						(* 1720: Bandklemmen links *)
						zyl_bandklemmen_li.fb.st_config.b_config_fertig := FALSE;
						zyl_bandklemmen_li.fb.st_config.b_endlage1_aktiv := FALSE;
						zyl_bandklemmen_li.fb.st_config.b_endlage2_aktiv := FALSE;
						zyl_bandklemmen_li.fb.st_config.b_sensor1_aktiv := FALSE;
						zyl_bandklemmen_li.fb.st_config.b_sensor2_aktiv := FALSE;
						zyl_bandklemmen_li.fb.st_config.i16_gruppe := 1;
						zyl_bandklemmen_li.fb.st_config.i16_identnummer := 3;
						zyl_bandklemmen_li.fb.st_config.i16_meld_startindex := 2040;
						zyl_bandklemmen_li.fb.st_config.str_beschreibung := ' ';
						zyl_bandklemmen_li.fb.st_config.str_instanz_name := 'Bandklemmen links';
						zyl_bandklemmen_li.fb.st_config.str_zylinder_typ := '1V0E_NO';
						zyl_bandklemmen_li.fb.st_config.t_ein_aus_fahrzeit := t#0ms;
						zyl_bandklemmen_li.fb.st_config.t_ueberwachungszeit := t#500ms;
						zyl_bandklemmen_li.fb.st_config.i16_tzk_faktor_ausfahren := 100;
						zyl_bandklemmen_li.fb.st_config.i16_tzk_faktor_einfahren := 100;
						zyl_bandklemmen_li.fb.st_config.b_config_fertig := TRUE;
						(* 1720: Bandklemmen rechts *)
						zyl_bandklemmen_re.fb.st_config.b_config_fertig := FALSE;
						zyl_bandklemmen_re.fb.st_config.b_endlage1_aktiv := FALSE;
						zyl_bandklemmen_re.fb.st_config.b_endlage2_aktiv := FALSE;
						zyl_bandklemmen_re.fb.st_config.b_sensor1_aktiv := FALSE;
						zyl_bandklemmen_re.fb.st_config.b_sensor2_aktiv := FALSE;
						zyl_bandklemmen_re.fb.st_config.i16_gruppe := 1;
						zyl_bandklemmen_re.fb.st_config.i16_identnummer := 4;
						zyl_bandklemmen_re.fb.st_config.i16_meld_startindex := 2060;
						zyl_bandklemmen_re.fb.st_config.str_beschreibung := ' ';
						zyl_bandklemmen_re.fb.st_config.str_instanz_name := 'Bandklemmen rechts';
						zyl_bandklemmen_re.fb.st_config.str_zylinder_typ := '1V0E_NO';
						zyl_bandklemmen_re.fb.st_config.t_ein_aus_fahrzeit := t#0ms;
						zyl_bandklemmen_re.fb.st_config.t_ueberwachungszeit := t#500ms;
						zyl_bandklemmen_re.fb.st_config.i16_tzk_faktor_ausfahren := 100;
						zyl_bandklemmen_re.fb.st_config.i16_tzk_faktor_einfahren := 100;
						zyl_bandklemmen_re.fb.st_config.b_config_fertig := TRUE;
				
					BANDWECHSLER_V2:
						;

					SERVO:
						;
				END_CASE;
		ELSE
			b_config_fertig := FALSE;
		END_IF

	RASTERFOLIE:
		;
END_CASE
END_PROGRAM

(* POU Maschine1720/ST_Bandeinzug_Kontroller_1720, ST *)
PROGRAM ST_Bandeinzug_Kontroller_1720
VAR_INPUT
	st_config							: struct_config;
	st_ctrl_in							: struct_ctrl_in;
END_VAR
VAR_IN_OUT
	st_visu							: struct_visu;
END_VAR
VAR_OUTPUT
	st_ctrl_out						: struct_ctrl_out;
END_VAR
VAR
	fb_ton_wz						: TON;
	fb_ton_uez						: TON;
	fb_ton_quitt						: TON;
	fb_state_entry						: ST_StateEntry;
	e_ls_bandende_re				AT %I* : BOOL;
	e_ls_bandende_li					AT %I* : BOOL;

	fb_r_trig_vorschubkontrolle_li		: R_TRIG;
	fb_f_trig_vorschubkontrolle_li		: F_TRIG;
	fb_r_trig_nocke_einzug				: R_TRIG;
	fb_f_trig_nocke_einzug				: F_TRIG;
	b_hm_pos_flanke_vorschub_li		: BOOL := FALSE;
	b_hm_neg_flanke_vorschub_li		: BOOL := FALSE;
	sm_fehler_bandvorschub_li			: BOOL := FALSE;
	fb_r_trig_vorschubkontrolle_re		: R_TRIG;
	fb_f_trig_vorschubkontrolle_re		: F_TRIG;
	b_hm_pos_flanke_vorschub_re		: BOOL := FALSE;
	b_hm_neg_flanke_vorschub_re		: BOOL := FALSE;
	sm_fehler_bandvorschub_re			: BOOL := FALSE;
	sm_keine_busverbindung			: BOOL := FALSE;

	e_wc_state							AT %I* : BOOL;	(* 0=Data valid, 1=Data invalid *)
	e_gls_bandvorschubkontrolle_li		AT %I* : BOOL;
	e_gls_bandvorschubkontrolle_re		AT %I* : BOOL;
END_VAR
(* Zeiten *)
fb_ton_wz(IN:= , PT:= , Q=>  , ET=> );
fb_ton_uez(IN:= , PT:= , Q=>  , ET=> );
fb_ton_quitt(IN:= , PT:= t#100ms, Q=> , ET=> );

(* Flanken *)
fb_f_trig_vorschubkontrolle_li(CLK:= e_gls_bandvorschubkontrolle_li, Q=> );
fb_r_trig_vorschubkontrolle_li(CLK:= e_gls_bandvorschubkontrolle_li, Q=> );
fb_f_trig_nocke_einzug(CLK:= nockenschaltwerk_bestueckachse.fb.arr_spur[SP_PNEUMATIKBANDEINZUG_GLS], Q=> );
fb_r_trig_nocke_einzug(CLK:= nockenschaltwerk_bestueckachse.fb.arr_spur[SP_PNEUMATIKBANDEINZUG_GLS], Q=> );
fb_f_trig_vorschubkontrolle_re(CLK:= e_gls_bandvorschubkontrolle_re, Q=> );
fb_r_trig_vorschubkontrolle_re(CLK:= e_gls_bandvorschubkontrolle_re, Q=> );

(*neue Haltezylinder für Bandklemmeinzug*)
(*bei Steuerung Ein oben bei Steuerung Aus wird selbständig über Federkraft geklemmt*)
IF ST_Safetyprogramm.se_steuerung_ein THEN
	zyl_bawe_halter_li.st_ctrl.in.b_einfahren := TRUE;
	zyl_bawe_halter_re.st_ctrl.in.b_einfahren := TRUE;
END_IF

(* Toplevel *)
IF fb_state_entry.i16_next_step > INIT AND fb_state_entry.i16_next_step < FEHLER THEN
	IF fb_state_entry.i16_next_step < STOP THEN
		IF st_ctrl_in.b_stop THEN
			fb_state_entry.i16_next_step := STOP;
		END_IF
	END_IF
	(* Allgemeine Fehler *)
	IF	NOT gst_datensatz.st_md.b_wt_transport_simulation AND
		(zyl_bandfaenger_li.st_ctrl.out.b_fehler OR
		zyl_bandklemmen_li.st_ctrl.out.b_fehler OR
		zyl_bandfaenger_re.st_ctrl.out.b_fehler OR
		zyl_bandklemmen_re.st_ctrl.out.b_fehler OR
		zyl_bawe_halter_li.st_ctrl.out.b_fehler OR
		zyl_bawe_halter_re.st_ctrl.out.b_fehler)
		THEN
			fb_state_entry.i16_next_step := FEHLER;
	(* Zylinder im Handbetrieb *)
	ELSIF	 gi16_betriebsart = HAND AND (
			(st_visu.st_zyl.i16_nr_zyl_im_handbetrieb = zyl_bandfaenger_li.fb.st_config.i16_identnummer OR
			st_visu.st_zyl.i16_nr_zyl_im_handbetrieb = zyl_bandfaenger_li.fb.st_config.i16_identnummer OR
			st_visu.st_zyl.i16_nr_zyl_im_handbetrieb = zyl_bandfaenger_re.fb.st_config.i16_identnummer OR
			st_visu.st_zyl.i16_nr_zyl_im_handbetrieb = zyl_bandklemmen_re.fb.st_config.i16_identnummer OR
			st_visu.st_zyl.i16_nr_zyl_im_handbetrieb = zyl_bawe_halter_li.fb.st_config.i16_identnummer OR
			st_visu.st_zyl.i16_nr_zyl_im_handbetrieb = zyl_bawe_halter_re.fb.st_config.i16_identnummer))
			THEN
				fb_state_entry.i16_next_step := FEHLER;
	END_IF
END_IF

(* ======================================Schrittkette======================================== *)
fb_state_entry(
	i16_next_step:= ,
	i16_pos:= 1,
	s_debugtext:= ,
	E=> ,
	X=> , 
	i16_step=> ,
	i16_last_step=> );

CASE fb_state_entry.i16_step OF
(*=======================================================*)
	INIT_OBJ:
		IF st_config.b_config_fertig THEN
			fb_state_entry.i16_next_step := INIT;
		END_IF

(*=======================================================*)
	INIT:
		IF fb_state_entry.E THEN
			fb_ton_wz.IN := FALSE;
			fb_ton_uez.IN := FALSE;
			fb_ton_quitt.IN := FALSE;
			st_ctrl_out.b_fehler := FALSE;
			st_ctrl_out.b_bereit := FALSE;
			st_ctrl_out.b_fertig := FALSE;
			zyl_bandfaenger_li.st_ctrl.in.b_ausfahren := FALSE;
			zyl_bandfaenger_li.st_ctrl.in.b_einfahren := FALSE;
			 zyl_bandklemmen_li.st_ctrl.in.b_ausfahren := FALSE;
			 zyl_bandklemmen_li.st_ctrl.in.b_einfahren := FALSE;
			zyl_bandfaenger_re.st_ctrl.in.b_ausfahren := FALSE;
			zyl_bandfaenger_re.st_ctrl.in.b_einfahren := FALSE;
			 zyl_bandklemmen_re.st_ctrl.in.b_ausfahren := FALSE;
			 zyl_bandklemmen_re.st_ctrl.in.b_einfahren := FALSE;
			sm_fehler_bandvorschub_li := FALSE;
			sm_fehler_bandvorschub_re := FALSE;
			sm_keine_busverbindung := FALSE;
		END_IF

		(*-----------------------Weiterschaltbedingungen----------------------------*)
		IF st_ctrl_in.b_init THEN
			zyl_bandfaenger_li.st_ctrl.in.b_quittieren := FALSE;
			zyl_bandklemmen_li.st_ctrl.in.b_quittieren := FALSE;
			zyl_bandfaenger_re.st_ctrl.in.b_quittieren := FALSE;
			zyl_bandklemmen_re.st_ctrl.in.b_quittieren := FALSE;
			zyl_bawe_halter_li.st_ctrl.in.b_quittieren := FALSE;
			zyl_bawe_halter_re.st_ctrl.in.b_quittieren := FALSE;
			IF gst_datensatz.st_md.b_wt_transport_simulation THEN
				fb_state_entry.i16_next_step := BEREIT;
			ELSE
				(*fb_state_entry.i16_next_step := 20; Bei nächster TSM-Änderung bitte aktivieren*)
				fb_state_entry.i16_next_step := BEREIT;
			END_IF
		END_IF

(*=======================================================*)
	20: (* Prüfe, ob Busverbindung vorhanden ist *)

		(*-----------------------Weiterschaltbedingungen----------------------------*)
		IF e_wc_state THEN	(* Prüfe Busverbindung ( 0=Data valid, 1=Data invalid )*)
			sm_keine_busverbindung := TRUE;
			fb_state_entry.i16_next_step := FEHLER;
		ELSE
			fb_state_entry.i16_next_step := BEREIT;
		END_IF

(*=======================================================*)
	BEREIT:
		IF fb_state_entry.E THEN
			st_ctrl_out.b_bereit := TRUE;
		END_IF

		(*-----------------------Weiterschaltbedingungen----------------------------*)
		CASE gst_datensatz.st_wkz.i16_typ_bandeinzug OF

			STANDARD_2FACH_V2:
				fb_state_entry.i16_next_step := 200;


			BANDWECHSLER_V2:
				(* Den Bandwechsler gibt es nur bei BSH1700 *)
				;
		END_CASE;

(*===========================Bandvorschub mit GLS-Kontrolle============================*)
	200:	(* Warte auf Vorschubnocke  und Freigabe von der Bestückachse *)
		(* Die Freigabe erfolgt nur im normalen Produktionsablauf; nicht bei Bandwechsel, Einfädeln, ... da hier keine Überwachung erfolgen soll. *)

		(*-----------------------Weiterschaltbedingungen----------------------------*)
		IF fb_r_trig_nocke_einzug.Q AND gi16_betriebsart <> HAND AND st_ctrl_in.b_freigabe THEN
			b_hm_pos_flanke_vorschub_li := FALSE;
			b_hm_neg_flanke_vorschub_li := FALSE;
			b_hm_pos_flanke_vorschub_re := FALSE;
			b_hm_neg_flanke_vorschub_re := FALSE;
			fb_state_entry.i16_next_step := 210;
		END_IF

(*=======================================================*)
	210:	(* Band links bzw. rechts wird vorgeschoben *)
		(* Vorschubkontrolle durch positive Flanke *)
		IF fb_r_trig_vorschubkontrolle_li.Q THEN
			b_hm_pos_flanke_vorschub_li := TRUE;
		END_IF
		IF fb_r_trig_vorschubkontrolle_re.Q THEN
			b_hm_pos_flanke_vorschub_re := TRUE;
		END_IF
		(* Vorschubkontrolle durch negative Flanke *)
		IF fb_f_trig_vorschubkontrolle_li.Q THEN
			b_hm_neg_flanke_vorschub_li := TRUE;
		END_IF
		IF fb_f_trig_vorschubkontrolle_re.Q THEN
			b_hm_neg_flanke_vorschub_re := TRUE;
		END_IF


		(*-----------------------Weiterschaltbedingungen----------------------------*)
		IF fb_f_trig_nocke_einzug.Q THEN
			IF 	b_hm_pos_flanke_vorschub_li AND b_hm_neg_flanke_vorschub_li AND
				b_hm_pos_flanke_vorschub_re AND b_hm_neg_flanke_vorschub_re
				THEN
					fb_state_entry.i16_next_step := 200;
			ELSE
				IF NOT b_hm_pos_flanke_vorschub_li OR NOT b_hm_neg_flanke_vorschub_li THEN
					sm_fehler_bandvorschub_li := TRUE;
				END_IF
				IF NOT b_hm_pos_flanke_vorschub_re OR NOT b_hm_neg_flanke_vorschub_re THEN
					sm_fehler_bandvorschub_re := TRUE;
				END_IF
				fb_state_entry.i16_next_step := FEHLER;
			END_IF
		ELSIF gi16_betriebsart = HAND THEN
			fb_state_entry.i16_next_step := 200;
		END_IF

(*=======================================================*)
	FEHLER:
		IF fb_state_entry.E THEN
			st_ctrl_out.b_fehler := TRUE;
			fb_ton_quitt.IN := FALSE;
			zyl_bandfaenger_li.st_ctrl.in.b_quittieren := FALSE;
			zyl_bandklemmen_li.st_ctrl.in.b_quittieren := FALSE;
			zyl_bandfaenger_re.st_ctrl.in.b_quittieren := FALSE;
			zyl_bandklemmen_re.st_ctrl.in.b_quittieren := FALSE;
			zyl_bawe_halter_li.st_ctrl.in.b_quittieren := FALSE;
			zyl_bawe_halter_re.st_ctrl.in.b_quittieren := FALSE;
		END_IF

		(*-----------------------Weiterschaltbedingungen----------------------------*)
		IF st_ctrl_in.b_quitt AND NOT fb_state_entry.E THEN
			st_ctrl_out.b_fehler := FALSE;
			zyl_bandfaenger_li.st_ctrl.in.b_quittieren := TRUE;
			zyl_bandklemmen_li.st_ctrl.in.b_quittieren := TRUE;
			zyl_bandfaenger_re.st_ctrl.in.b_quittieren := TRUE;
			zyl_bandklemmen_re.st_ctrl.in.b_quittieren := TRUE;
			zyl_bawe_halter_li.st_ctrl.in.b_quittieren := TRUE;
			zyl_bawe_halter_re.st_ctrl.in.b_quittieren := TRUE;
			fb_ton_quitt.IN := TRUE;
		END_IF

		IF fb_ton_quitt.Q THEN
			fb_ton_quitt.IN := FALSE;
			fb_state_entry.i16_next_step := INIT;
		END_IF

(*=======================================================*)
	STOP:
		IF fb_state_entry.E THEN
			fb_ton_quitt.IN := FALSE;
			zyl_bandfaenger_li.st_ctrl.in.b_quittieren := FALSE;
			zyl_bandklemmen_li.st_ctrl.in.b_quittieren := FALSE;
			zyl_bandfaenger_re.st_ctrl.in.b_quittieren := FALSE;
			zyl_bandklemmen_re.st_ctrl.in.b_quittieren := FALSE;
			zyl_bawe_halter_li.st_ctrl.in.b_quittieren := FALSE;
			zyl_bawe_halter_re.st_ctrl.in.b_quittieren := FALSE;
		END_IF

		(*-----------------------Weiterschaltbedingungen----------------------------*)
		IF st_ctrl_in.b_quitt AND NOT fb_state_entry.E THEN
			fb_ton_quitt.IN := TRUE;
			zyl_bandfaenger_li.st_ctrl.in.b_quittieren := TRUE;
			zyl_bandklemmen_li.st_ctrl.in.b_quittieren := TRUE;
			zyl_bandfaenger_re.st_ctrl.in.b_quittieren := TRUE;
			zyl_bandklemmen_re.st_ctrl.in.b_quittieren := TRUE;
			zyl_bawe_halter_li.st_ctrl.in.b_quittieren := TRUE;
			zyl_bawe_halter_re.st_ctrl.in.b_quittieren := TRUE;
		END_IF

		IF fb_ton_quitt.Q THEN
			fb_ton_quitt.IN := FALSE;
			fb_state_entry.i16_next_step := INIT;
		END_IF
END_CASE

fb_state_entry(
	i16_next_step:= , 
	i16_pos:= 2,
	s_debugtext:= ,
	E=> , 
	X=> , 
	i16_step=> ,
	i16_last_step=> );

IF st_config.b_config_fertig THEN
	(* Fehlermeldungen und Betriebsmeldungen ab dem Startindex in die globalen Meldungsarrays schreiben *)
	garr_stoermeldungen[st_config.i16_meld_startindex + 0] := FALSE;(* belegt  durch Bandeinzugskontroller 1700 *)
	garr_stoermeldungen[st_config.i16_meld_startindex + 1] := sm_fehler_bandvorschub_li;
	garr_stoermeldungen[st_config.i16_meld_startindex + 2] := sm_fehler_bandvorschub_re;
	garr_stoermeldungen[st_config.i16_meld_startindex + 3] := sm_keine_busverbindung;
	garr_stoermeldungen[st_config.i16_meld_startindex + 4] := FALSE;
	garr_stoermeldungen[st_config.i16_meld_startindex + 5] := FALSE;
	garr_stoermeldungen[st_config.i16_meld_startindex + 6] := FALSE;
	garr_stoermeldungen[st_config.i16_meld_startindex + 7] := FALSE;
	garr_stoermeldungen[st_config.i16_meld_startindex + 8] := FALSE;
	garr_stoermeldungen[st_config.i16_meld_startindex + 9] := FALSE;
	garr_stoermeldungen[st_config.i16_meld_startindex + 10] := FALSE;
	garr_stoermeldungen[st_config.i16_meld_startindex + 11] := FALSE;
	garr_stoermeldungen[st_config.i16_meld_startindex + 12] := FALSE;
	garr_stoermeldungen[st_config.i16_meld_startindex + 13] := FALSE;
	garr_stoermeldungen[st_config.i16_meld_startindex + 14] := FALSE;
	garr_stoermeldungen[st_config.i16_meld_startindex + 15] := FALSE;
	garr_stoermeldungen[st_config.i16_meld_startindex + 16] := FALSE;
	garr_stoermeldungen[st_config.i16_meld_startindex + 17] := FALSE;
	garr_stoermeldungen[st_config.i16_meld_startindex + 18] := FALSE;
	garr_stoermeldungen[st_config.i16_meld_startindex + 19] := FALSE;
	
	garr_betriebsmeldungen[st_config.i16_meld_startindex + 0] := FALSE;
	garr_betriebsmeldungen[st_config.i16_meld_startindex + 1] := FALSE;
	garr_betriebsmeldungen[st_config.i16_meld_startindex + 2] := FALSE;
	garr_betriebsmeldungen[st_config.i16_meld_startindex + 3] := FALSE;
	garr_betriebsmeldungen[st_config.i16_meld_startindex + 4] := FALSE;
	garr_betriebsmeldungen[st_config.i16_meld_startindex + 5] := FALSE;
	garr_betriebsmeldungen[st_config.i16_meld_startindex + 6] := FALSE;
	garr_betriebsmeldungen[st_config.i16_meld_startindex + 7] := FALSE;
	garr_betriebsmeldungen[st_config.i16_meld_startindex + 8] := FALSE;
	garr_betriebsmeldungen[st_config.i16_meld_startindex + 9] := FALSE;
	garr_betriebsmeldungen[st_config.i16_meld_startindex + 10] := FALSE;
	garr_betriebsmeldungen[st_config.i16_meld_startindex + 11] := FALSE;
	garr_betriebsmeldungen[st_config.i16_meld_startindex + 12] := FALSE;
	garr_betriebsmeldungen[st_config.i16_meld_startindex + 13] := FALSE;
	garr_betriebsmeldungen[st_config.i16_meld_startindex + 14] := FALSE;
	garr_betriebsmeldungen[st_config.i16_meld_startindex + 15] := FALSE;
	garr_betriebsmeldungen[st_config.i16_meld_startindex + 16] := FALSE;
	garr_betriebsmeldungen[st_config.i16_meld_startindex + 17] := FALSE;
	garr_betriebsmeldungen[st_config.i16_meld_startindex + 18] := FALSE;
	garr_betriebsmeldungen[st_config.i16_meld_startindex + 19] := FALSE;
END_IF
END_PROGRAM

(* POU MAINs/MAIN_STANDARD, ST *)
PROGRAM MAIN_STANDARD
VAR
END_VAR
CASE gst_datensatz.st_md.i16_typ_zelle OF
	KEINE_ZELLE:
		;
	BESTUECKZELLE_1700:
		IF visu.s_akt_sprache <> 'en' THEN
			ST_AutoCheckIn( i_IntervalDay:=7 );
		END_IF
		ST_SaveAndLoad();
		ST_Datainit_Stationen();
		ST_Datainit_Achsen();

		ST_EthercatDiag();

		(* Grundmaschine *)
		EtherCatDiag[1]( );
		EtherCatDiag[1].st_config.b_station_aktiv := TRUE;

		(* Hublift links *)
		EtherCatDiag[2]( );
		EtherCatDiag[2].st_config.b_station_aktiv := gst_datensatz.st_md.b_hublift_links_aktiv;

		(* Hublift rechts *)
		EtherCatDiag[3]( );
		EtherCatDiag[3].st_config.b_station_aktiv := gst_datensatz.st_md.b_hublift_rechts_aktiv;

		(* Bandeinzug *)
		(* Bandeinzug nicht aufrufen, weil in allen TSM der Mulitpol A170 für die Rasterfolie drin ist und dieser
		in keinem normalen Bandeinzug
		Bei normalem Bandeinzug kommt immer Fehler Busverbindung *)
		(*EtherCatDiag[4]( );
		EtherCatDiag[4].st_config.b_station_aktiv := NOT gst_datensatz.st_md.b_wt_transport_simulation;*)

		ST_UPS(st_config:= UPS.st_config,
			st_ctrl_in:= UPS.st_ctrl.in,
			b_Ups := TRUE,
			st_ctrl_out=> UPS.st_ctrl.out);

		ST_RoutingBackpanel(
			st_config:= routing_backpanel.st_config,
			st_ctrl_in:= routing_backpanel.st_ctrl.in,
			st_ctrl_out=> routing_backpanel.st_ctrl.out);

		ST_MotionFunctionPoints(
			st_ctrl_in:= edit_mfps.st_ctrl.in,
			st_ctrl_out=> edit_mfps.st_ctrl.out);

		ST_Schreibe_Persistente_Daten(
			bExecute:= ,
			bQuit:= ,
			t_schreibintervall:= t#60s,
			b_steuerung_ein:= ST_Safetyprogramm.se_steuerung_ein,
			bBusy=> ,
			bError=> ,
			nErrId=> );

		ST_System_DateAndTime();

		betriebsstundenzaehler.fb(
			b_eingekuppelt:= (ST_Z_Achse.fb_state_entry.i16_step > BEREIT AND ST_Z_Achse.fb_state_entry.i16_step < HALT) AND (gi16_betriebsart = AUTO),
			b_reset:= ,
			i32_betriebssekundenzaehler_in:= gst_datensatz.st_md.i32_betriebssekundenzaehler,
			i32_betriebssekundenzaehler=> gst_datensatz.st_md.i32_betriebssekundenzaehler);

		ST_Tuerverriegelung(
			e_quittiertaste:= ST_Safetyprogramm.se_quittiertaste);

		ST_LampeMaterialMangel(b_materialmangel:=  );

		ST_Zylinder();

		ST_start_OSK(bExecute:= ST_Safetyprogramm.se_quittiertaste);

		ST_Euchner_Handbedienpult();

		ST_TippTasten(
			i16_akt_stufe:= ,
			b_initialisierungsphase:= ,
			b_einfaedeln_aktiv:= ,
			st_visu:= visu,
			st_visu_hinten:= visu_hinten);

		ST_Betriebsarten(st_config:= betriebsarten.st_config);

		(* Übernahme der Daten aus der Datenbank: Beladen und Abgabe greifen dann auf diese Konfiguration zu *)
		wt_transport_kontroller.st_config.b_station_aktiv := gst_datensatz.st_md.b_wt_transport_aktiv;
		wt_transport_kontroller.st_config.b_station_in_simulation := gst_datensatz.st_md.b_wt_transport_simulation;

		ST_WT_Transport_Kontroller(
			st_config:= wt_transport_kontroller.st_config,
			st_ctrl_in:= wt_transport_kontroller.st_ctrl.in,
			st_visu:= visu,
			st_ctrl_out=> wt_transport_kontroller.st_ctrl.out);

		(* Aktivierung durch den Kontroller *)
		wt_transport_abgabe.st_config.b_station_aktiv := gst_datensatz.st_md.b_wt_transport_aktiv;
		wt_transport_abgabe.st_config.b_station_in_simulation := gst_datensatz.st_md.b_wt_transport_simulation;

		ST_WT_Transport_Abgabe(
			st_config:= wt_transport_abgabe.st_config,
			st_ctrl_in:= wt_transport_abgabe.st_ctrl.in,
			e_station_nachher_in_erlaubnis:= ,
			e_station_nachher_in_angekommen:= ,
			st_visu:= wt_transport_abgabe.st_visu,
			st_ctrl_out=> wt_transport_abgabe.st_ctrl.out,
			a_station_nachher_out_anforderung=> a_smema_station_nachher_out_anforderung,
			a_station_nachher_out_abgegeben=> a_smema_station_nachher_out_abgegeben);

		hublift_rechts.st_config.b_station_aktiv := gst_datensatz.st_md.b_hublift_rechts_aktiv;
		hublift_rechts.st_config.b_station_in_simulation := gst_datensatz.st_md.b_hublift_rechts_simulation;

		ST_Hublift_rechts(
			st_config:= hublift_rechts.st_config,
			st_ctrl_in:= hublift_rechts.st_ctrl.in,
			e_station_vorher_in_anforderung	:= ,
			e_station_vorher_in_abgegeben:= ,
			st_visu:= hublift_rechts.st_visu,
			st_ctrl_out=> hublift_rechts.st_ctrl.out,
			a_station_vorher_out_erlaubnis=> ,
			a_station_vorher_out_angekommen=> );
		IF hublift_rechts.st_config.b_station_aktiv OR hublift_rechts.st_config.b_station_in_simulation THEN
			ST_Hublift_rechts.e_station_vorher_in_abgegeben := ST_WT_Transport_Abgabe.a_station_nachher_out_abgegeben;
			ST_Hublift_rechts.e_station_vorher_in_anforderung := ST_WT_Transport_Abgabe.a_station_nachher_out_anforderung;
			ST_WT_Transport_Abgabe.e_station_nachher_in_angekommen := ST_Hublift_rechts.a_station_vorher_out_angekommen;
			ST_WT_Transport_Abgabe.e_station_nachher_in_erlaubnis := ST_Hublift_rechts.a_station_vorher_out_erlaubnis;
		ELSE
			ST_WT_Transport_Abgabe.e_station_nachher_in_angekommen := e_smema_station_nachher_in_angekommen;
			ST_WT_Transport_Abgabe.e_station_nachher_in_erlaubnis := e_smema_station_nachher_in_erlaubnis;
		END_IF

		balluff_tag_reader.fb(
			st_config:= balluff_tag_reader.fb.st_config,
			i16_addresse:= ,
			i16_anzahl_byte:= ,
			s_schreib_daten:= ,
			st_ctrl_in:= balluff_tag_reader.st_ctrl.in,
			s_lese_daten=> ,
			st_ctrl_out=> balluff_tag_reader.st_ctrl.out);

		barcode.fb(
			st_config:= barcode.fb.st_config,
			st_barcode_daten := gst_barcode_daten,
			b_steuerung_ein := ST_Safetyprogramm.se_steuerung_ein,
			b_bandende_links := ST_Bandwechsel_Kontroller.e_ls_bandende_li ,
			b_bandende_rechts := ST_Bandwechsel_Kontroller.e_ls_bandende_re,
			b_bandende_1720 := ST_Bandeinzug_Kontroller_1720.e_ls_bandende_li,
			b_band_nicht_gescannt=> ST_LampeMaterialMangel.b_materialmangel[5]);

		visu_hinten.in.bandfreigabe[0] := gst_barcode_daten.b_band_rechts_ok;
		visu_hinten.in.bandfreigabe[1] := gst_barcode_daten.b_band_links_ok;
		visu_hinten.in.band_ID[0] := gst_barcode_daten.b_band_ID_rechts_ok;
		visu_hinten.in.band_ID[1] := gst_barcode_daten.b_band_ID_links_ok;

		ST_VisuRouter();

		ST_Message_Produktion();

		ST_Bestueckachse(
			st_config_achse:= axis_bestueckachse.st_config,
			st_ctrl_in:= axis_bestueckachse.st_ctrl.in,
			e_steuerung_ein:= ST_Safetyprogramm.se_steuerung_ein,
			e_ba_mit_bedingungen:= ST_Safetyprogramm.se_ba_mit_bedingungen,
			e_tuere_vorne_offen:= ST_Safetyprogramm.se_tuere_vorne_offen,
			e_tuere_hinten_offen:= ST_Safetyprogramm.se_tuere_hinten_offen,
			st_visu:= axis_bestueckachse.st_visu,
			st_ctrl_out=> axis_bestueckachse.st_ctrl.out);

		ST_Z_Achse(
			st_config_achse:= axis_z_achse.st_config,
			st_ctrl_in:= axis_z_achse.st_ctrl.in,
			e_steuerung_ein:= ST_Safetyprogramm.se_steuerung_ein,
			e_ba_mit_bedingungen:= ST_Safetyprogramm.se_ba_mit_bedingungen,
			e_tuere_vorne_offen:= ST_Safetyprogramm.se_tuere_vorne_offen,
			e_tuere_hinten_offen:= ST_Safetyprogramm.se_tuere_hinten_offen,
			st_visu:= axis_z_achse.st_visu,
			st_ctrl_out=> axis_z_achse.st_ctrl.out,
			t_Z_Achse_ausfahren=>visu.ST_Service.t_Z_Achse_ausfahren,
			t_Bestueckung=>visu.ST_Service.t_Bestueckung,
			t_Z_Achse_einfahren=>visu.ST_Service.t_Z_Achse_einfahren);

		ST_TouchProbe();

		ST_Y_Achse(
			st_config_achse:= axis_y_achse.st_config,
			st_ctrl_in:= axis_y_achse.st_ctrl.in,
			e_steuerung_ein:= ST_Safetyprogramm.se_steuerung_ein,
			e_ba_mit_bedingungen:= ST_Safetyprogramm.se_ba_mit_bedingungen,
			e_tuere_vorne_offen:= ST_Safetyprogramm.se_tuere_vorne_offen,
			e_tuere_hinten_offen:= ST_Safetyprogramm.se_tuere_hinten_offen,
			e_not_steu_tuer_schutz_ok:= ,
			st_visu:= axis_y_achse.st_visu,
			st_ctrl_out=> axis_y_achse.st_ctrl.out);


		ST_Gesamthubzaehler();

		IF gst_Datensatz.st_md.b_anwahl_transport_achse THEN

			ST_WT_Transport_Achse(
				st_config_achse:= axis_transport_wt_achse.st_config,
				st_ctrl_in:= axis_transport_wt_achse.st_ctrl.in,
				e_steuerung_ein:= ST_Safetyprogramm.se_steuerung_ein,
				e_ba_mit_bedingungen:= ST_Safetyprogramm.se_ba_mit_bedingungen,
				e_tuere_vorne_offen:= ST_Safetyprogramm.se_tuere_vorne_offen,
				e_tuere_hinten_offen:= ST_Safetyprogramm.se_tuere_hinten_offen,
				st_visu:= axis_transport_wt_achse.st_visu,
				st_ctrl_out=> axis_transport_wt_achse.st_ctrl.out);

			wt_transport_warteposition_1700.st_config.b_station_aktiv := gst_datensatz.st_md.b_wt_transport_aktiv;
			wt_transport_warteposition_1700.st_config.b_station_in_simulation := gst_datensatz.st_md.b_wt_transport_simulation;

			ST_WT_Transport_Warteposition_1700(
				st_config:= wt_transport_warteposition_1700.st_config,
				st_ctrl_in:= wt_transport_warteposition_1700.st_ctrl.in,
				e_station_vorher_in_anforderung	:= ,
				e_station_vorher_in_abgegeben:= ,
				st_visu:= wt_transport_warteposition_1700.st_visu,
				st_ctrl_out=> wt_transport_warteposition_1700.st_ctrl.out,
				a_station_vorher_out_erlaubnis=> a_smema_station_vorher_out_erlaubnis,
				a_station_vorher_out_angekommen=> a_smema_station_vorher_out_angekommen);
	
			wt_transport_beladen_achse_1700.st_config.b_station_aktiv := gst_datensatz.st_md.b_wt_transport_aktiv;
			wt_transport_beladen_achse_1700.st_config.b_station_in_simulation := gst_datensatz.st_md.b_wt_transport_simulation;
	
			ST_WT_Transport_Beladen_Achse_1700(
				st_config:= wt_transport_beladen_achse_1700.st_config,
				st_ctrl_in:= wt_transport_beladen_achse_1700.st_ctrl.in,
				e_wt_im_aktionsfeld := balluff_tag_reader.fb.e_tag_im_aktionsfeld,
				st_visu:= wt_transport_beladen_achse_1700.st_visu,
				st_ctrl_out=> wt_transport_beladen_achse_1700.st_ctrl.out,
				t_WT_WechselZeit=>visu.ST_Service.t_WT_wechsel,
				t_traegerwechselzeit=>visu.ST_Service.t_traegerwechselzeit,
				t_Zentrierer_ausfahren=>visu.ST_Service.t_Zentrierer_ausfahren,
				t_Zentrierer_einfahren=>visu.ST_Service.t_Zentrierer_einfahren,
				t_komplett_zyklus=>visu.ST_Service.t_komplett_zyklus,);

		ELSE
			(* Aktivierung durch den Kontroller *)
			wt_transport_beladen.st_config.b_station_aktiv := gst_datensatz.st_md.b_wt_transport_aktiv;
			wt_transport_beladen.st_config.b_station_in_simulation := gst_datensatz.st_md.b_wt_transport_simulation;
	
			ST_WT_Transport_Beladen(
				st_config:= wt_transport_beladen.st_config,
				st_ctrl_in:= wt_transport_beladen.st_ctrl.in,
				e_station_vorher_in_anforderung	:= ,
				e_station_vorher_in_abgegeben:= ,
				st_visu:= wt_transport_beladen.st_visu,
				st_ctrl_out=> wt_transport_beladen.st_ctrl.out,
				a_station_vorher_out_erlaubnis=> a_smema_station_vorher_out_erlaubnis,
				a_station_vorher_out_angekommen=> a_smema_station_vorher_out_angekommen,
				t_WT_WechselZeit=>visu.ST_Service.t_WT_wechsel,
				t_traegerwechselzeit=>visu.ST_Service.t_traegerwechselzeit,
				t_Zentrierer_ausfahren=>visu.ST_Service.t_Zentrierer_ausfahren,
				t_Zentrierer_einfahren=>visu.ST_Service.t_Zentrierer_einfahren,
				t_komplett_zyklus=>visu.ST_Service.t_komplett_zyklus,);
		END_IF

		hublift_links.st_config.b_station_aktiv := gst_datensatz.st_md.b_hublift_links_aktiv;
		hublift_links.st_config.b_station_in_simulation := gst_datensatz.st_md.b_hublift_links_simulation;

		ST_Hublift_links(
			st_config:= hublift_links.st_config,
			st_ctrl_in:= hublift_links.st_ctrl.in,
			e_station_nachher_in_erlaubnis:= ,
			e_station_nachher_in_angekommen:= ,
			st_visu:= hublift_links.st_visu,
			st_ctrl_out=> hublift_links.st_ctrl.out,
			a_station_nachher_out_anforderung=> ,
			a_station_nachher_out_abgegeben=> );
		IF hublift_links.st_config.b_station_aktiv OR hublift_links.st_config.b_station_in_simulation THEN
			IF gst_Datensatz.st_md.b_anwahl_transport_achse THEN
				ST_WT_Transport_Warteposition_1700.e_station_vorher_in_abgegeben := ST_Hublift_links.a_station_nachher_out_abgegeben;
				ST_WT_Transport_Warteposition_1700.e_station_vorher_in_anforderung := ST_Hublift_links.a_station_nachher_out_anforderung;
				ST_Hublift_links.e_station_nachher_in_angekommen := ST_WT_Transport_Warteposition_1700.a_station_vorher_out_angekommen;
				ST_Hublift_links.e_station_nachher_in_erlaubnis := ST_WT_Transport_Warteposition_1700.a_station_vorher_out_erlaubnis;
			ELSE
				ST_WT_Transport_Beladen.e_station_vorher_in_abgegeben := ST_Hublift_links.a_station_nachher_out_abgegeben;
				ST_WT_Transport_Beladen.e_station_vorher_in_anforderung := ST_Hublift_links.a_station_nachher_out_anforderung;
				ST_Hublift_links.e_station_nachher_in_angekommen := ST_WT_Transport_Beladen.a_station_vorher_out_angekommen;
				ST_Hublift_links.e_station_nachher_in_erlaubnis := ST_WT_Transport_Beladen.a_station_vorher_out_erlaubnis;
			END_IF
		ELSE
			IF gst_Datensatz.st_md.b_anwahl_transport_achse THEN
				ST_WT_Transport_Warteposition_1700.e_station_vorher_in_abgegeben := e_smema_station_vorher_in_abgegeben;
				ST_WT_Transport_Warteposition_1700.e_station_vorher_in_anforderung := e_smema_station_vorher_in_anforderung;
			ELSE
				ST_WT_Transport_Beladen.e_station_vorher_in_abgegeben := e_smema_station_vorher_in_abgegeben;
				ST_WT_Transport_Beladen.e_station_vorher_in_anforderung := e_smema_station_vorher_in_anforderung;
			END_IF
		END_IF

		ST_Stoerungen_Quitt_1700(
			st_config:= stoerungen_quittieren.st_config,
			st_ctrl_in:= stoerungen_quittieren.st_ctrl.in,
			st_visu:= visu,
			st_visu_hinten:= visu_hinten,
			st_ctrl_out=> stoerungen_quittieren.st_ctrl.out,
			b_lampe_stoerung=> ST_Betriebsfreigaben.b_lampe_stoerung,
			b_lampe_produktion=> ST_Betriebsfreigaben.b_lampe_produktion);

		ST_Bandwechsel_Kontroller(
			st_config:= bandwechsel_kontroller.st_config,
			st_ctrl_in:= bandwechsel_kontroller.st_ctrl.in,
			st_visu:= visu,
			b_materialmangel=> ST_LampeMaterialMangel.b_materialmangel[3],
			st_ctrl_out=> bandwechsel_kontroller.st_ctrl.out);

		ST_Haspel_Kontroller_2H(
			t_abschaltzeit_motor:= haspel_kontroller.t_abschaltzeit_motor,
			b_drehrichtung_antrieb_links := gst_datensatz.st_wkz.b_laufrichtung_haspel_links,
			st_config:= haspel_kontroller.st_config,
			e_druckwaechter:= ST_Betriebsfreigaben.e_druckwaechter,
			e_steuerung_ein:= ST_Safetyprogramm.se_steuerung_ein,
			st_ctrl_in:= haspel_kontroller.st_ctrl.in,
			haspel1_ctrl_in:= haspel_li.st_ctrl.out,
			haspel2_ctrl_in:= haspel_re.st_ctrl.out,
			st_visu:= haspel_kontroller.st_visu,
			st_ctrl_out=> haspel_kontroller.st_ctrl.out,
			haspel1_ctrl_out=> haspel_li.st_ctrl.in,
			haspel2_ctrl_out=> haspel_re.st_ctrl.in,
			b_materialmangel_bandende=> ST_LampeMaterialMangel.b_materialmangel[0]);

		Haspel_Li.fb(
			t_wartezeit_bandende:= t#5s,
			b_bandende_Bandeinzug := ST_Bandwechsel_Kontroller.e_ls_bandende_li ,
			b_band_ok := gst_barcode_daten.b_band_links_ok AND gst_barcode_daten.b_band_ID_links_ok,
			st_config:= Haspel_Li.fb.st_config,
			st_ctrl_in:= Haspel_Li.st_ctrl.in,
			st_visu := Haspel_Li.st_visu,
			st_zyl_heben:= zyl_haspel_li_heben,
			st_zyl_abspulen:= zyl_haspel_li_abspulen,
			st_zyl_sperren:= zyl_haspel_li_sperren,
			st_ctrl_out=> Haspel_Li.st_ctrl.out);

		Haspel_Re.fb(
			t_wartezeit_bandende:= t#5s,
			b_bandende_Bandeinzug := ST_Bandwechsel_Kontroller.e_ls_bandende_re ,
			b_band_ok := gst_barcode_daten.b_band_rechts_ok AND gst_barcode_daten.b_band_ID_rechts_ok ,
			st_config:= Haspel_Re.fb.st_config,
			st_ctrl_in:= Haspel_Re.st_ctrl.in,
			st_visu := Haspel_Re.st_visu,
			st_zyl_heben:= zyl_haspel_re_heben,
			st_zyl_abspulen:= zyl_haspel_re_abspulen,
			st_zyl_sperren:= zyl_haspel_re_sperren,
			st_ctrl_out=> Haspel_Re.st_ctrl.out);

		IF gst_datensatz.st_md.b_auswahlSpruehoeler THEN
			ST_Menzel_Spruehoeler(
				st_config:= bandspruehoeler.st_config,
				st_ctrl_in:= bandspruehoeler.st_ctrl.in,
				lr_achse_position:= bestueckachse.NcToPlc.ModuloActPos,
				e_steuerung_ein:= ST_Safetyprogramm.se_steuerung_ein,
				e_druckwaechter:= ST_Betriebsfreigaben.e_druckwaechter,
				st_ctrl_out =>bandspruehoeler.st_ctrl.out,
				b_oelmangel=> ST_LampeMaterialMangel.b_materialmangel[1]);
		ELSE
			ST_BandoelerZylinder(
					st_config:= bandspruehoeler.st_config,
					st_ctrl_in:= bandspruehoeler.st_ctrl.in,
					lr_achse_position:= bestueckachse.NcToPlc.ModuloActPos,
					e_steuerung_ein:= ST_Safetyprogramm.se_steuerung_ein,
					e_druckwaechter:= ST_Betriebsfreigaben.e_druckwaechter,
					st_ctrl_out =>bandspruehoeler.st_ctrl.out,
					b_oelmangel=> ST_LampeMaterialMangel.b_materialmangel[1]);
		END_IF

		ST_Lesen_Schreiben_Tag(
			st_config:= Lesen_Schreiben_Tag.st_config,
			st_ctrl_in:= Lesen_Schreiben_Tag.st_ctrl.in,
			st_ctrl_out=> Lesen_Schreiben_Tag.st_ctrl.out);

		ST_Anwahl_Bandeinzug();
		ST_Scope();

	BESTUECKZELLE_1720:
		ST_AutoCheckIn( i_IntervalDay:=7 );
		ST_SaveAndLoad();
		ST_Datainit_Stationen();
		ST_Datainit_Achsen();

		ST_EthercatDiag();

		(* Grundmaschine *)
		EtherCatDiag[1]( );
		EtherCatDiag[1].st_config.b_station_aktiv := TRUE;

		(* Hublift links *)
		EtherCatDiag[2]( );
		EtherCatDiag[2].st_config.b_station_aktiv := gst_datensatz.st_md.b_hublift_links_aktiv;

		(* Hublift rechts *)
		EtherCatDiag[3]( );
		EtherCatDiag[3].st_config.b_station_aktiv := gst_datensatz.st_md.b_hublift_rechts_aktiv;

		(* Bandeinzug *)
		EtherCatDiag[4]( );
		EtherCatDiag[4].st_config.b_station_aktiv := NOT gst_datensatz.st_md.b_wt_transport_simulation;

		ST_UPS(st_config:= UPS.st_config,
			st_ctrl_in:= UPS.st_ctrl.in,
			b_Ups := TRUE,
			st_ctrl_out=> UPS.st_ctrl.out);

		ST_RoutingBackpanel(
			st_config:= routing_backpanel.st_config,
			st_ctrl_in:= routing_backpanel.st_ctrl.in,
			st_ctrl_out=> routing_backpanel.st_ctrl.out);

		ST_MotionFunctionPoints(
			st_ctrl_in:= edit_mfps.st_ctrl.in,
			st_ctrl_out=> edit_mfps.st_ctrl.out);

		ST_Schreibe_Persistente_Daten(
			bExecute:= ,
			bQuit:= ,
			t_schreibintervall:= t#60s,
			b_steuerung_ein:= ST_Safetyprogramm.se_steuerung_ein,
			bBusy=> ,
			bError=> ,
			nErrId=> );

		ST_System_DateAndTime();

		betriebsstundenzaehler.fb(
			b_eingekuppelt:= (ST_Z_Achse.fb_state_entry.i16_step > BEREIT AND ST_Z_Achse.fb_state_entry.i16_step < HALT) AND (gi16_betriebsart = AUTO),
			b_reset:= ,
			i32_betriebssekundenzaehler_in:= gst_datensatz.st_md.i32_betriebssekundenzaehler,
			i32_betriebssekundenzaehler=> gst_datensatz.st_md.i32_betriebssekundenzaehler);

		ST_Tuerverriegelung(
			e_quittiertaste:= ST_Safetyprogramm.se_quittiertaste);

		ST_LampeMaterialMangel(b_materialmangel:=  );

		ST_Zylinder();

		ST_start_OSK(bExecute:= ST_Safetyprogramm.se_quittiertaste);

		ST_Euchner_Handbedienpult();

		ST_TippTasten(
			i16_akt_stufe:= ,
			b_initialisierungsphase:= ,
			b_einfaedeln_aktiv:= ,
			st_visu:= visu,
			st_visu_hinten:= visu_hinten);

		ST_Betriebsarten(st_config:= betriebsarten.st_config);

		(* Übernahme der Daten aus der Datenbank: Beladen und Abgabe greifen dann auf diese Konfiguration zu *)
		wt_transport_kontroller.st_config.b_station_aktiv := gst_datensatz.st_md.b_wt_transport_aktiv;
		wt_transport_kontroller.st_config.b_station_in_simulation := gst_datensatz.st_md.b_wt_transport_simulation;

		ST_WT_Transport_Kontroller(
			st_config:= wt_transport_kontroller.st_config,
			st_ctrl_in:= wt_transport_kontroller.st_ctrl.in,
			st_visu:= visu,
			st_ctrl_out=> wt_transport_kontroller.st_ctrl.out);

		(* Aktivierung durch den Kontroller *)
		wt_transport_abgabe.st_config.b_station_aktiv := gst_datensatz.st_md.b_wt_transport_aktiv;
		wt_transport_abgabe.st_config.b_station_in_simulation := gst_datensatz.st_md.b_wt_transport_simulation;

		ST_WT_Transport_Abgabe(
			st_config:= wt_transport_abgabe.st_config,
			st_ctrl_in:= wt_transport_abgabe.st_ctrl.in,
			e_station_nachher_in_erlaubnis:= ,
			e_station_nachher_in_angekommen:= ,
			st_visu:= wt_transport_abgabe.st_visu,
			st_ctrl_out=> wt_transport_abgabe.st_ctrl.out,
			a_station_nachher_out_anforderung=> a_smema_station_nachher_out_anforderung,
			a_station_nachher_out_abgegeben=> a_smema_station_nachher_out_abgegeben);

		hublift_rechts.st_config.b_station_aktiv := gst_datensatz.st_md.b_hublift_rechts_aktiv;
		hublift_rechts.st_config.b_station_in_simulation := gst_datensatz.st_md.b_hublift_rechts_simulation;

		ST_Hublift_rechts(
			st_config:= hublift_rechts.st_config,
			st_ctrl_in:= hublift_rechts.st_ctrl.in,
			e_station_vorher_in_anforderung	:= ,
			e_station_vorher_in_abgegeben:= ,
			st_visu:= hublift_rechts.st_visu,
			st_ctrl_out=> hublift_rechts.st_ctrl.out,
			a_station_vorher_out_erlaubnis=> ,
			a_station_vorher_out_angekommen=> );
		IF hublift_rechts.st_config.b_station_aktiv OR hublift_rechts.st_config.b_station_in_simulation THEN
			ST_Hublift_rechts.e_station_vorher_in_abgegeben := ST_WT_Transport_Abgabe.a_station_nachher_out_abgegeben;
			ST_Hublift_rechts.e_station_vorher_in_anforderung := ST_WT_Transport_Abgabe.a_station_nachher_out_anforderung;
			ST_WT_Transport_Abgabe.e_station_nachher_in_angekommen := ST_Hublift_rechts.a_station_vorher_out_angekommen;
			ST_WT_Transport_Abgabe.e_station_nachher_in_erlaubnis := ST_Hublift_rechts.a_station_vorher_out_erlaubnis;
		ELSE
			ST_WT_Transport_Abgabe.e_station_nachher_in_angekommen := e_smema_station_nachher_in_angekommen;
			ST_WT_Transport_Abgabe.e_station_nachher_in_erlaubnis := e_smema_station_nachher_in_erlaubnis;
		END_IF

		balluff_tag_reader.fb(
			st_config:= balluff_tag_reader.fb.st_config,
			i16_addresse:= ,
			i16_anzahl_byte:= ,
			s_schreib_daten:= ,
			st_ctrl_in:= balluff_tag_reader.st_ctrl.in,
			s_lese_daten=> ,
			st_ctrl_out=> balluff_tag_reader.st_ctrl.out);

		barcode.fb(
			st_config:= barcode.fb.st_config,
			st_barcode_daten := gst_barcode_daten,
			b_steuerung_ein := ST_Safetyprogramm.se_steuerung_ein,
			b_bandende_links := ST_Bandeinzug_Kontroller_1720.e_ls_bandende_li ,
			b_bandende_rechts := ST_Bandeinzug_Kontroller_1720.e_ls_bandende_re,
			b_bandende_1720 := ST_Bandeinzug_Kontroller_1720.e_ls_bandende_li OR ST_Bandeinzug_Kontroller_1720.e_ls_bandende_re,
			b_band_nicht_gescannt=> ST_LampeMaterialMangel.b_materialmangel[5]);

		visu_hinten.in.bandfreigabe[0] := gst_barcode_daten.b_band_rechts_ok;
		visu_hinten.in.bandfreigabe[1] := gst_barcode_daten.b_band_links_ok;
		visu_hinten.in.band_ID[0] := gst_barcode_daten.b_band_ID_rechts_ok;
		visu_hinten.in.band_ID[1] := gst_barcode_daten.b_band_ID_links_ok;

		ST_VisuRouter();

		ST_Message_Produktion();

		ST_Bestueckachse(
			st_config_achse:= axis_bestueckachse.st_config,
			st_ctrl_in:= axis_bestueckachse.st_ctrl.in,
			e_steuerung_ein:= ST_Safetyprogramm.se_steuerung_ein,
			e_ba_mit_bedingungen:= ST_Safetyprogramm.se_ba_mit_bedingungen,
			e_tuere_vorne_offen:= ST_Safetyprogramm.se_tuere_vorne_offen,
			e_tuere_hinten_offen:= ST_Safetyprogramm.se_tuere_hinten_offen,
			st_visu:= axis_bestueckachse.st_visu,
			st_ctrl_out=> axis_bestueckachse.st_ctrl.out);

		ST_Z_Achse(
			st_config_achse:= axis_z_achse.st_config,
			st_ctrl_in:= axis_z_achse.st_ctrl.in,
			e_steuerung_ein:= ST_Safetyprogramm.se_steuerung_ein,
			e_ba_mit_bedingungen:= ST_Safetyprogramm.se_ba_mit_bedingungen,
			e_tuere_vorne_offen:= ST_Safetyprogramm.se_tuere_vorne_offen,
			e_tuere_hinten_offen:= ST_Safetyprogramm.se_tuere_hinten_offen,
			st_visu:= axis_z_achse.st_visu,
			st_ctrl_out=> axis_z_achse.st_ctrl.out,
			t_Z_Achse_ausfahren=>visu.ST_Service.t_Z_Achse_ausfahren,
			t_Bestueckung=>visu.ST_Service.t_Bestueckung,
			t_Z_Achse_einfahren=>visu.ST_Service.t_Z_Achse_einfahren);

		ST_TouchProbe();

		ST_Gesamthubzaehler();

		(* Aktivierung durch den Kontroller *)
		wt_transport_warteposition_1720.st_config.b_station_aktiv := gst_datensatz.st_md.b_wt_transport_aktiv;
		wt_transport_warteposition_1720.st_config.b_station_in_simulation := gst_datensatz.st_md.b_wt_transport_simulation;

		ST_WT_Transport_Warteposition_1720(
			st_config:= wt_transport_warteposition_1720.st_config,
			st_ctrl_in:= wt_transport_warteposition_1720.st_ctrl.in,
			e_station_vorher_in_anforderung	:= ,
			e_station_vorher_in_abgegeben:= ,
			st_visu:= wt_transport_warteposition_1720.st_visu,
			st_ctrl_out=> wt_transport_warteposition_1720.st_ctrl.out,
			a_station_vorher_out_erlaubnis=> a_smema_station_vorher_out_erlaubnis,
			a_station_vorher_out_angekommen=> a_smema_station_vorher_out_angekommen);

		(* Aktivierung durch den Kontroller *)
		wt_transport_beladen_1720.st_config.b_station_aktiv := gst_datensatz.st_md.b_wt_transport_aktiv;
		wt_transport_beladen_1720.st_config.b_station_in_simulation := gst_datensatz.st_md.b_wt_transport_simulation;

		ST_WT_Transport_Beladen_1720(
			st_config:= wt_transport_beladen_1720.st_config,
			st_ctrl_in:= wt_transport_beladen_1720.st_ctrl.in,
			st_visu:= wt_transport_beladen_1720.st_visu,
			st_ctrl_out=> wt_transport_beladen_1720.st_ctrl.out,
			t_WT_WechselZeit=>visu.ST_Service.t_WT_wechsel,
			t_traegerwechselzeit=>visu.ST_Service.t_traegerwechselzeit,
			t_Zentrierer_ausfahren=>visu.ST_Service.t_Zentrierer_ausfahren,
			t_Zentrierer_einfahren=>visu.ST_Service.t_Zentrierer_einfahren,
			t_komplett_zyklus=>visu.ST_Service.t_komplett_zyklus,);

		hublift_links.st_config.b_station_aktiv := gst_datensatz.st_md.b_hublift_links_aktiv;
		hublift_links.st_config.b_station_in_simulation := gst_datensatz.st_md.b_hublift_links_simulation;

		ST_Hublift_links(
			st_config:= hublift_links.st_config,
			st_ctrl_in:= hublift_links.st_ctrl.in,
			e_station_nachher_in_erlaubnis:= ,
			e_station_nachher_in_angekommen:= ,
			st_visu:= hublift_links.st_visu,
			st_ctrl_out=> hublift_links.st_ctrl.out,
			a_station_nachher_out_anforderung=> ,
			a_station_nachher_out_abgegeben=> );
		IF hublift_links.st_config.b_station_aktiv OR hublift_links.st_config.b_station_in_simulation THEN
			ST_Hublift_links.e_station_nachher_in_angekommen := ST_WT_Transport_Warteposition_1720.a_station_vorher_out_angekommen;
			ST_Hublift_links.e_station_nachher_in_erlaubnis := ST_WT_Transport_Warteposition_1720.a_station_vorher_out_erlaubnis;
			ST_WT_Transport_Warteposition_1720.e_station_vorher_in_abgegeben := ST_Hublift_links.a_station_nachher_out_abgegeben;
			ST_WT_Transport_Warteposition_1720.e_station_vorher_in_anforderung := ST_Hublift_links.a_station_nachher_out_anforderung;
		ELSE
			ST_WT_Transport_Warteposition_1720.e_station_vorher_in_abgegeben := e_smema_station_vorher_in_abgegeben;
			ST_WT_Transport_Warteposition_1720.e_station_vorher_in_anforderung := e_smema_station_vorher_in_anforderung;
		END_IF

		ST_Stoerungen_Quitt_1720(
			st_config:= stoerungen_quittieren.st_config,
			st_ctrl_in:= stoerungen_quittieren.st_ctrl.in,
			st_visu:= visu,
			st_visu_hinten:= visu_hinten,
			st_ctrl_out=> stoerungen_quittieren.st_ctrl.out,
			b_lampe_stoerung=> ST_Betriebsfreigaben.b_lampe_stoerung,
			b_lampe_produktion=> ST_Betriebsfreigaben.b_lampe_produktion);

		ST_Haspel_Kontroller_2H(
			t_abschaltzeit_motor:= haspel_kontroller.t_abschaltzeit_motor,
			b_drehrichtung_antrieb_links := gst_datensatz.st_wkz.b_laufrichtung_haspel_links,
			st_config:= haspel_kontroller.st_config,
			e_druckwaechter:= ST_Betriebsfreigaben.e_druckwaechter,
			e_steuerung_ein:= ST_Safetyprogramm.se_steuerung_ein,
			st_ctrl_in:= haspel_kontroller.st_ctrl.in,
			haspel1_ctrl_in:= haspel_li.st_ctrl.out,
			haspel2_ctrl_in:= haspel_re.st_ctrl.out,
			st_visu:= haspel_kontroller.st_visu,
			st_ctrl_out=> haspel_kontroller.st_ctrl.out,
			haspel1_ctrl_out=> haspel_li.st_ctrl.in,
			haspel2_ctrl_out=> haspel_re.st_ctrl.in,
			b_materialmangel_bandende=> ST_LampeMaterialMangel.b_materialmangel[0]);

		Haspel_Li.fb(
			t_wartezeit_bandende:= t#5s,
			b_bandende_Bandeinzug := ST_Bandwechsel_Kontroller.e_ls_bandende_li ,
			st_config:= Haspel_Li.fb.st_config,
			st_ctrl_in:= Haspel_Li.st_ctrl.in,
			st_visu := Haspel_Li.st_visu,
			st_zyl_heben:= zyl_haspel_li_heben,
			st_zyl_abspulen:= zyl_haspel_li_abspulen,
			st_zyl_sperren:= zyl_haspel_li_sperren,
			st_ctrl_out=> Haspel_Li.st_ctrl.out);

		Haspel_Re.fb(
			t_wartezeit_bandende:= t#5s,
			b_bandende_Bandeinzug := ST_Bandwechsel_Kontroller.e_ls_bandende_re ,
			st_config:= Haspel_Re.fb.st_config,
			st_ctrl_in:= Haspel_Re.st_ctrl.in,
			st_visu := Haspel_Re.st_visu,
			st_zyl_heben:= zyl_haspel_re_heben,
			st_zyl_abspulen:= zyl_haspel_re_abspulen,
			st_zyl_sperren:= zyl_haspel_re_sperren,
			st_ctrl_out=> Haspel_Re.st_ctrl.out);

		ST_Menzel_Spruehoeler(
			st_config:= bandspruehoeler.st_config,
			st_ctrl_in:= bandspruehoeler.st_ctrl.in,
			lr_achse_position:= bestueckachse.NcToPlc.ModuloActPos,
			e_steuerung_ein:= ST_Safetyprogramm.se_steuerung_ein,
			e_druckwaechter:= ST_Betriebsfreigaben.e_druckwaechter,
			st_ctrl_out =>bandspruehoeler.st_ctrl.out,
			b_oelmangel=> ST_LampeMaterialMangel.b_materialmangel[1]);

		ST_AbfallBlasluft(
			b_wkz_blasluft_aktiv:= gst_datensatz.st_wkz.b_wkz_blasluft_aktiv);

		ST_Lesen_Schreiben_Tag(
			st_config:= Lesen_Schreiben_Tag.st_config,
			st_ctrl_in:= Lesen_Schreiben_Tag.st_ctrl.in,
			st_ctrl_out=> Lesen_Schreiben_Tag.st_ctrl.out);

		ST_Anwahl_Bandeinzug();
		ST_Scope();

	RASTERFOLIE:
		ST_AutoCheckIn( i_IntervalDay:=7 );
		ST_SaveAndLoad();
		ST_Datainit_Stationen();
		ST_Datainit_Achsen();

		ST_EthercatDiag();

		(* Grundmaschine *)
		EtherCatDiag[1]( );
		EtherCatDiag[1].st_config.b_station_aktiv := TRUE;

		(* Hublift links *)
		EtherCatDiag[2]( );
		EtherCatDiag[2].st_config.b_station_aktiv := gst_datensatz.st_md.b_hublift_links_aktiv;

		(* Hublift rechts *)
		EtherCatDiag[3]( );
		EtherCatDiag[3].st_config.b_station_aktiv := gst_datensatz.st_md.b_hublift_rechts_aktiv;

		(* Bandeinzug *)
		EtherCatDiag[4]( );
		EtherCatDiag[4].st_config.b_station_aktiv := NOT gst_datensatz.st_md.b_wt_transport_simulation;

		ST_UPS(st_config:= UPS.st_config,
			st_ctrl_in:= UPS.st_ctrl.in,
			b_Ups := TRUE,
			st_ctrl_out=> UPS.st_ctrl.out);

		ST_RoutingBackpanel(
			st_config:= routing_backpanel.st_config,
			st_ctrl_in:= routing_backpanel.st_ctrl.in,
			st_ctrl_out=> routing_backpanel.st_ctrl.out);


		ST_MotionFunctionPoints(
			st_ctrl_in:= edit_mfps.st_ctrl.in,
			st_ctrl_out=> edit_mfps.st_ctrl.out);

		ST_Schreibe_Persistente_Daten(
			bExecute:= ,
			bQuit:= ,
			t_schreibintervall:= t#60s,
			b_steuerung_ein:= ST_Safetyprogramm.se_steuerung_ein,
			bBusy=> ,
			bError=> ,
			nErrId=> );

		ST_System_DateAndTime();

		betriebsstundenzaehler.fb(
			b_eingekuppelt:= (ST_Z_Achse.fb_state_entry.i16_step > BEREIT AND ST_Z_Achse.fb_state_entry.i16_step < HALT) AND (gi16_betriebsart = AUTO),
			b_reset:= ,
			i32_betriebssekundenzaehler_in:= gst_datensatz.st_md.i32_betriebssekundenzaehler,
			i32_betriebssekundenzaehler=> gst_datensatz.st_md.i32_betriebssekundenzaehler);

		ST_Tuerverriegelung(
			e_quittiertaste:= ST_Safetyprogramm.se_quittiertaste);

		ST_LampeMaterialMangel(b_materialmangel:=  );

		ST_Zylinder();

		ST_start_OSK(bExecute:= ST_Safetyprogramm.se_quittiertaste);

		ST_Euchner_Handbedienpult();

		ST_TippTasten(
			i16_akt_stufe:= ,
			b_initialisierungsphase:= ,
			b_einfaedeln_aktiv:= ,
			st_visu:= visu,
			st_visu_hinten:= visu_hinten);

		ST_Betriebsarten(st_config:= betriebsarten.st_config);

		(* Übernahme der Daten aus der Datenbank: Beladen und Abgabe greifen dann auf diese Konfiguration zu *)
		wt_transport_kontroller.st_config.b_station_aktiv := gst_datensatz.st_md.b_wt_transport_aktiv;
		wt_transport_kontroller.st_config.b_station_in_simulation := gst_datensatz.st_md.b_wt_transport_simulation;

		ST_WT_Transport_Kontroller(
			st_config:= wt_transport_kontroller.st_config,
			st_ctrl_in:= wt_transport_kontroller.st_ctrl.in,
			st_visu:= visu,
			st_ctrl_out=> wt_transport_kontroller.st_ctrl.out);

		(* Aktivierung durch den Kontroller *)
		wt_transport_abgabe.st_config.b_station_aktiv := gst_datensatz.st_md.b_wt_transport_aktiv;
		wt_transport_abgabe.st_config.b_station_in_simulation := gst_datensatz.st_md.b_wt_transport_simulation;

		ST_WT_Transport_Abgabe(
			st_config:= wt_transport_abgabe.st_config,
			st_ctrl_in:= wt_transport_abgabe.st_ctrl.in,
			e_station_nachher_in_erlaubnis:= ,
			e_station_nachher_in_angekommen:= ,
			st_visu:= wt_transport_abgabe.st_visu,
			st_ctrl_out=> wt_transport_abgabe.st_ctrl.out,
			a_station_nachher_out_anforderung=> a_smema_station_nachher_out_anforderung,
			a_station_nachher_out_abgegeben=> a_smema_station_nachher_out_abgegeben);

		hublift_rechts.st_config.b_station_aktiv := gst_datensatz.st_md.b_hublift_rechts_aktiv;
		hublift_rechts.st_config.b_station_in_simulation := gst_datensatz.st_md.b_hublift_rechts_simulation;

		ST_Hublift_rechts(
			st_config:= hublift_rechts.st_config,
			st_ctrl_in:= hublift_rechts.st_ctrl.in,
			e_station_vorher_in_anforderung	:= ,
			e_station_vorher_in_abgegeben:= ,
			st_visu:= hublift_rechts.st_visu,
			st_ctrl_out=> hublift_rechts.st_ctrl.out,
			a_station_vorher_out_erlaubnis=> ,
			a_station_vorher_out_angekommen=> );
		IF hublift_rechts.st_config.b_station_aktiv OR hublift_rechts.st_config.b_station_in_simulation THEN
			ST_Hublift_rechts.e_station_vorher_in_abgegeben := ST_WT_Transport_Abgabe.a_station_nachher_out_abgegeben;
			ST_Hublift_rechts.e_station_vorher_in_anforderung := ST_WT_Transport_Abgabe.a_station_nachher_out_anforderung;
			ST_WT_Transport_Abgabe.e_station_nachher_in_angekommen := ST_Hublift_rechts.a_station_vorher_out_angekommen;
			ST_WT_Transport_Abgabe.e_station_nachher_in_erlaubnis := ST_Hublift_rechts.a_station_vorher_out_erlaubnis;
		ELSE
			ST_WT_Transport_Abgabe.e_station_nachher_in_angekommen := e_smema_station_nachher_in_angekommen;
			ST_WT_Transport_Abgabe.e_station_nachher_in_erlaubnis := e_smema_station_nachher_in_erlaubnis;
		END_IF

		balluff_tag_reader.fb(
			st_config:= balluff_tag_reader.fb.st_config,
			i16_addresse:= ,
			i16_anzahl_byte:= ,
			s_schreib_daten:= ,
			st_ctrl_in:= balluff_tag_reader.st_ctrl.in,
			s_lese_daten=> ,
			st_ctrl_out=> balluff_tag_reader.st_ctrl.out);

		barcode.fb(
			st_config:= barcode.fb.st_config,
			st_barcode_daten := gst_barcode_daten,
			b_steuerung_ein := ST_Safetyprogramm.se_steuerung_ein,
			b_bandende_links := ST_Bandwechsel_Kontroller.e_ls_bandende_li ,
			b_bandende_rechts := ST_Bandwechsel_Kontroller.e_ls_bandende_re,
			b_bandende_1720 := ST_Bandeinzug_Kontroller_1720.e_ls_bandende_li,
			b_band_nicht_gescannt=> ST_LampeMaterialMangel.b_materialmangel[5]);

		visu_hinten.in.bandfreigabe[0] := gst_barcode_daten.b_band_rechts_ok;
		visu_hinten.in.bandfreigabe[1] := gst_barcode_daten.b_band_links_ok;
		visu_hinten.in.band_ID[0] := gst_barcode_daten.b_band_ID_rechts_ok;
		visu_hinten.in.band_ID[1] := gst_barcode_daten.b_band_ID_links_ok;

		ST_VisuRouter();

		ST_Message_Produktion();

 		ST_Rafl_Stoerungen_Quitt(
			st_config:= stoerungen_quittieren.st_config,
			st_ctrl_in:= stoerungen_quittieren.st_ctrl.in,
			st_visu:= visu,
			st_visu_hinten:= visu_hinten,
			st_ctrl_out=> stoerungen_quittieren.st_ctrl.out,
			b_lampe_stoerung=> ST_Betriebsfreigaben.b_lampe_stoerung,
			b_lampe_produktion=> ST_Betriebsfreigaben.b_lampe_produktion);

		ST_Rasterfolienmontage(
			st_config:= rasterfolienmontage.st_config,
			st_ctrl_in:= rasterfolienmontage.st_ctrl.in,
			st_visu:= rasterfolienmontage.st_visu,
			st_ctrl_out=> rasterfolienmontage.st_ctrl.out);

		ST_Rasterfolieneinzug(
			st_config:= rasterfolieneinzug.st_config,
			st_ctrl_in:= rasterfolieneinzug.st_ctrl.in,
			st_visu:= rasterfolieneinzug.st_visu,
			st_ctrl_out=> rasterfolieneinzug.st_ctrl.out);

		ST_Bestueckachse(
			st_config_achse:= axis_bestueckachse.st_config,
			st_ctrl_in:= axis_bestueckachse.st_ctrl.in,
			e_steuerung_ein:= ST_Safetyprogramm.se_steuerung_ein,
			e_ba_mit_bedingungen:= ST_Safetyprogramm.se_ba_mit_bedingungen,
			e_tuere_vorne_offen:= ST_Safetyprogramm.se_tuere_vorne_offen,
			e_tuere_hinten_offen:= ST_Safetyprogramm.se_tuere_hinten_offen,
			st_visu:= axis_bestueckachse.st_visu,
			st_ctrl_out=> axis_bestueckachse.st_ctrl.out);

		ST_Z_Achse(
			st_config_achse:= axis_z_achse.st_config,
			st_ctrl_in:= axis_z_achse.st_ctrl.in,
			e_steuerung_ein:= ST_Safetyprogramm.se_steuerung_ein,
			e_ba_mit_bedingungen:= ST_Safetyprogramm.se_ba_mit_bedingungen,
			e_tuere_vorne_offen:= ST_Safetyprogramm.se_tuere_vorne_offen,
			e_tuere_hinten_offen:= ST_Safetyprogramm.se_tuere_hinten_offen,
			st_visu:= axis_z_achse.st_visu,
			st_ctrl_out=> axis_z_achse.st_ctrl.out,
			t_Z_Achse_ausfahren=>visu.ST_Service.t_Z_Achse_ausfahren,
			t_Bestueckung=>visu.ST_Service.t_Bestueckung,
			t_Z_Achse_einfahren=>visu.ST_Service.t_Z_Achse_einfahren);

		ST_Y_Achse(
			st_config_achse:= axis_y_achse.st_config,
			st_ctrl_in:= axis_y_achse.st_ctrl.in,
			e_steuerung_ein:= ST_Safetyprogramm.se_steuerung_ein,
			e_ba_mit_bedingungen:= ST_Safetyprogramm.se_ba_mit_bedingungen,
			e_tuere_vorne_offen:= ST_Safetyprogramm.se_tuere_vorne_offen,
			e_tuere_hinten_offen:= ST_Safetyprogramm.se_tuere_hinten_offen,
			e_not_steu_tuer_schutz_ok:= ,
			st_visu:= axis_y_achse.st_visu,
			st_ctrl_out=> axis_y_achse.st_ctrl.out);

		ST_Gesamthubzaehler();

		(* Aktivierung durch den Kontroller *)
		wt_transport_beladen.st_config.b_station_aktiv := gst_datensatz.st_md.b_wt_transport_aktiv;
		wt_transport_beladen.st_config.b_station_in_simulation := gst_datensatz.st_md.b_wt_transport_simulation;

		ST_WT_Transport_Beladen(
			st_config:= wt_transport_beladen.st_config,
			st_ctrl_in:= wt_transport_beladen.st_ctrl.in,
			e_station_vorher_in_anforderung	:= ,
			e_station_vorher_in_abgegeben:= ,
			st_visu:= wt_transport_beladen.st_visu,
			st_ctrl_out=> wt_transport_beladen.st_ctrl.out,
			a_station_vorher_out_erlaubnis=> a_smema_station_vorher_out_erlaubnis,
			a_station_vorher_out_angekommen=> a_smema_station_vorher_out_angekommen,
			t_WT_WechselZeit=>visu.ST_Service.t_WT_wechsel,
			t_traegerwechselzeit=>visu.ST_Service.t_traegerwechselzeit,
			t_Zentrierer_ausfahren=>visu.ST_Service.t_Zentrierer_ausfahren,
			t_Zentrierer_einfahren=>visu.ST_Service.t_Zentrierer_einfahren,
			t_komplett_zyklus=>visu.ST_Service.t_komplett_zyklus,);

		hublift_links.st_config.b_station_aktiv := gst_datensatz.st_md.b_hublift_links_aktiv;
		hublift_links.st_config.b_station_in_simulation := gst_datensatz.st_md.b_hublift_links_simulation;

		ST_Hublift_links(
			st_config:= hublift_links.st_config,
			st_ctrl_in:= hublift_links.st_ctrl.in,
			e_station_nachher_in_erlaubnis:= ,
			e_station_nachher_in_angekommen:= ,
			st_visu:= hublift_links.st_visu,
			st_ctrl_out=> hublift_links.st_ctrl.out,
			a_station_nachher_out_anforderung=> ,
			a_station_nachher_out_abgegeben=> );
		IF hublift_links.st_config.b_station_aktiv OR hublift_links.st_config.b_station_in_simulation THEN
			ST_Hublift_links.e_station_nachher_in_angekommen := ST_WT_Transport_Beladen.a_station_vorher_out_angekommen;
			ST_Hublift_links.e_station_nachher_in_erlaubnis := ST_WT_Transport_Beladen.a_station_vorher_out_erlaubnis;
			ST_WT_Transport_Beladen.e_station_vorher_in_abgegeben := ST_Hublift_links.a_station_nachher_out_abgegeben;
			ST_WT_Transport_Beladen.e_station_vorher_in_anforderung := ST_Hublift_links.a_station_nachher_out_anforderung;
		ELSE
			ST_WT_Transport_Beladen.e_station_vorher_in_abgegeben := e_smema_station_vorher_in_abgegeben;
			ST_WT_Transport_Beladen.e_station_vorher_in_anforderung := e_smema_station_vorher_in_anforderung;
		END_IF

		ST_Lesen_Schreiben_Tag(
			st_config:= Lesen_Schreiben_Tag.st_config,
			st_ctrl_in:= Lesen_Schreiben_Tag.st_ctrl.in,
			st_ctrl_out=> Lesen_Schreiben_Tag.st_ctrl.out);

		ST_Anwahl_Bandeinzug();
		ST_Scope();

		ST_TouchProbe();

		ST_Haspel_Kontroller_2H(
			t_abschaltzeit_motor:= haspel_kontroller.t_abschaltzeit_motor,
			b_drehrichtung_antrieb_links := gst_datensatz.st_wkz.b_laufrichtung_haspel_links,
			st_config:= haspel_kontroller.st_config,
			e_druckwaechter:= ST_Betriebsfreigaben.e_druckwaechter,
			e_steuerung_ein:= ST_Safetyprogramm.se_steuerung_ein,
			st_ctrl_in:= haspel_kontroller.st_ctrl.in,
			haspel1_ctrl_in:= haspel_li.st_ctrl.out,
			haspel2_ctrl_in:= haspel_re.st_ctrl.out,
			st_visu:= haspel_kontroller.st_visu,
			st_ctrl_out=> haspel_kontroller.st_ctrl.out,
			haspel1_ctrl_out=> haspel_li.st_ctrl.in,
			haspel2_ctrl_out=> haspel_re.st_ctrl.in,
			b_materialmangel_bandende=> ST_LampeMaterialMangel.b_materialmangel[0]);

		Haspel_Li.fb(
			t_wartezeit_bandende:= t#5s,
			b_bandende_Bandeinzug := ST_Bandwechsel_Kontroller.e_ls_bandende_li ,
			b_band_ok := gst_barcode_daten.b_band_links_ok AND gst_barcode_daten.b_band_ID_links_ok,
			st_config:= Haspel_Li.fb.st_config,
			st_ctrl_in:= Haspel_Li.st_ctrl.in,
			st_visu := Haspel_Li.st_visu,
			st_zyl_heben:= zyl_haspel_li_heben,
			st_zyl_abspulen:= zyl_haspel_li_abspulen,
			st_zyl_sperren:= zyl_haspel_li_sperren,
			st_ctrl_out=> Haspel_Li.st_ctrl.out);

		Haspel_Re.fb(
			t_wartezeit_bandende:= t#5s,
			b_bandende_Bandeinzug := ST_Bandwechsel_Kontroller.e_ls_bandende_re ,
			b_band_ok := gst_barcode_daten.b_band_rechts_ok AND gst_barcode_daten.b_band_ID_rechts_ok ,
			st_config:= Haspel_Re.fb.st_config,
			st_ctrl_in:= Haspel_Re.st_ctrl.in,
			st_visu := Haspel_Re.st_visu,
			st_zyl_heben:= zyl_haspel_re_heben,
			st_zyl_abspulen:= zyl_haspel_re_abspulen,
			st_zyl_sperren:= zyl_haspel_re_sperren,
			st_ctrl_out=> Haspel_Re.st_ctrl.out);

END_CASE
END_PROGRAM

(* POU EPT Lib/Daten/ST_AutoCheckIn, ST *)
PROGRAM ST_AutoCheckIn
VAR_INPUT
	st_ctrl_in				: struct_ctrl_in;
	fb_AutocheckinDaten	: FB_StartWinProcess;
	i_IntervalDay				: INT;		(*all  X Tagen, 0 = jeden Tag*)
END_VAR
VAR_OUTPUT
	st_ctrl_out				: struct_ctrl_out;
END_VAR
VAR
	fb_state_entry			:ST_StateEntry;
	fb_ton_quitt				:TON;

	str_uhrzeit				:STRING;
	i_DayOfYear			:DINT;
	s_infoFile				:STRING;
	s_ScriptFile				:STRING;

END_VAR

VAR CONSTANT
		s_AutoCheckInMDtxt				:STRING:=		'AutoCheckInMD.txt';
		s_AutoCheckInMDBat				:STRING:=		'AutoCheckInMD.bat';

END_VAR
(*======================================================
   FB: Start eines Win Prozess mit Prüfung 
 ------------------------------------------------------
   Auth: 		Werner Friedl   						 
   Date: 		19.02.2019   						     
   Rev.: 		1.0	
   Desc:		Mit diesem Programm Können Komponenten im Versdog automatisch eingecheckt werden.
			Für den Check in benötigt man einen Bat- Datei. Diese liegt im Projektverzeichniss "Tools" und 
			muss für jede Komponente erstellt werden.
			Wenn mehrere Komponeten Eingecheckt werden sollen muss der Schritt 110 bis 120 mehrfach
			ausgefühtr werden.

			- die Input Variable "i16_Intervall" legt den Seicherintervall in x Tagen fest.
			Wenn das Speichern nicht klappt, dann wird einen Tag später der nächste Versuch gemacht.

   Historie:   1.0

=======================================================*)

(* Zeiten *)
fb_ton_quitt(IN:= , PT:= t#100ms, Q=> , ET=> );

(* Tag im Jahr *)
i_DayOfYear:=F_GetDOYOfYearMonthDay( gst_system_time.wYear, gst_system_time.wMonth, gst_system_time.wDay );

fb_state_entry(i16_pos:= 1);

CASE fb_state_entry.i16_step OF

(*=======================================================*)
INIT_OBJ:

	(*-----------------------Weiterschaltbedingungen----------------------------*)
	IF	gst_datensatz.st_md.i16_typ_zelle <> KEINE_ZELLE AND
		gstr_uhrzeit <> '00:00:00' AND gstr_uhrzeit <> ''  THEN
		IF	gst_PersDaten.i_DayOfYearAutoCheckIn > i_DayOfYear THEN
			gst_PersDaten.i_DayOfYearAutoCheckIn:= i_DayOfYear;
		END_IF
			fb_state_entry.i16_next_step := 5;
	END_IF

(*=======================================================*)
5:
	IF fb_state_entry.E THEN
		str_uhrzeit:=gstr_uhrzeit;
		(*str_uhrzeit:=REPLACE (str_uhrzeit,'00',2,1);*)	(*nur in der Nacht sichern*)
	END_IF

	(*-----------------------Weiterschaltbedingungen----------------------------*)
	IF 	fb_state_entry.fb_ton_Step.ET > t#59s THEN
		IF	gst_PersDaten.i_DayOfYearAutoCheckIn + i_IntervalDay < i_DayOfYear  THEN
			fb_state_entry.i16_next_step:=110;		(*gleich sicher, da das letzte Sichern zu lange her ist*)
		ELSE
			fb_state_entry.i16_next_step:=INIT;
		END_IF
	END_IF

(*=======================================================*)
INIT:
	IF fb_state_entry.E THEN
		fb_ton_quitt.IN := FALSE;
		st_ctrl_out.b_fehler := FALSE;
		st_ctrl_out.b_gestoppt := FALSE;
		st_ctrl_out.b_bereit := FALSE;
		st_ctrl_out.b_fertig := FALSE;
		st_ctrl_out.b_busy := FALSE;
	END_IF

	(*-----------------------Weiterschaltbedingungen----------------------------*)
	fb_state_entry.i16_next_step := BEREIT;

(*=======================================================*)
BEREIT: fb_state_entry.s_debugtext:='warte auf Start';

	IF fb_state_entry.E THEN
		st_ctrl_out.b_bereit:=TRUE;
	END_IF

	(*-----------------------Weiterschaltbedingungen----------------------------*)
	IF 	str_uhrzeit=gstr_uhrzeit AND
		(gst_PersDaten.i_DayOfYearAutoCheckIn + i_IntervalDay) <= i_DayOfYear THEN
		fb_state_entry.i16_next_step:=110;
	END_IF

	IF fb_state_entry.X THEN
		st_ctrl_out.b_busy:=TRUE;
		st_ctrl_out.b_bereit := FALSE;
		st_ctrl_out.b_fertig := FALSE;
	END_IF

(*=======================================================*)
110:  fb_state_entry.s_debugtext:='Start Autocheckin';

	IF fb_state_entry.E THEN
		s_infoFile:=s_AutoCheckInMDtxt;
		s_ScriptFile:=s_AutoCheckInMDBat;
		fb_AutocheckinDaten.st_ctrl_in.b_start:=TRUE;
	END_IF

	(*-----------------------Weiterschaltbedingungen----------------------------*)
	IF	fb_AutocheckinDaten.st_ctrl_out.b_busy THEN
		fb_state_entry.i16_next_step:=120;
	ELSIF	fb_state_entry.fb_ton_Step.ET > t#15s THEN
		fb_state_entry.i16_next_step:=FEHLER;
	END_IF

(*=======================================================*)
120:  fb_state_entry.s_debugtext:='Warte auf fertig Autocheckin';

	(*-----------------------Weiterschaltbedingungen----------------------------*)
	IF	fb_AutocheckinDaten.st_ctrl_out.b_fertig THEN
		fb_state_entry.i16_next_step:=200;
	ELSIF
		fb_state_entry.fb_ton_Step.ET > t#59s OR
		fb_AutocheckinDaten.st_ctrl_out.b_fehler THEN
		fb_state_entry.i16_next_step:=FEHLER;
		gst_PersDaten.i_DayOfYearAutoCheckIn:=i_DayOfYear - i_IntervalDay+1; (*bei einem Fehler wird die nächst Sicherung einen Tag später nochmal gemacht*)
	END_IF

(*=======================================================*)
200:  fb_state_entry.s_debugtext:='Ende';

	(*-----------------------Weiterschaltbedingungen----------------------------*)
	fb_state_entry.i16_next_step:=BEREIT;
	gst_PersDaten.i_DayOfYearAutoCheckIn:=i_DayOfYear;
	IF fb_state_entry.X THEN
		st_ctrl_out.b_busy:=FALSE;
		st_ctrl_out.b_fertig := TRUE;
	END_IF

(*=======================================================*)
STOP, FEHLER:
	IF fb_state_entry.E THEN
		st_ctrl_out.b_fehler := fb_state_entry.i16_step = FEHLER;
		st_ctrl_out.b_gestoppt := fb_state_entry.i16_step = STOP;
		fb_ton_quitt.IN := FALSE;
		st_ctrl_out.b_busy:=FALSE;
		st_ctrl_out.b_fertig:=FALSE;
		fb_ton_quitt.IN := TRUE;				(*quttiert sich selbst*)
	END_IF

	(*-----------------------Weiterschaltbedingungen----------------------------*)
	IF 	st_ctrl_in.b_quitt THEN
		fb_ton_quitt.IN := TRUE;
	END_IF

	IF fb_ton_quitt.Q THEN
		fb_ton_quitt.IN := FALSE;
		st_ctrl_out.b_fehler := FALSE;
		fb_state_entry.i16_next_step := INIT;
	END_IF

END_CASE

fb_state_entry(i16_pos:= 2 );
st_ctrl_in:=st_ctrl_in_empty;


(*Aufrufe======================================================*)
fb_AutocheckinDaten(
	s_path:= 			s_tools_path,								(*Verzeichnis der bat,vbs und Prüf- Datei*)
	s_info_file:=			CONCAT(s_tools_path,s_infoFile) ,			(*Datei in der die Prüfung landet*)
	s_script:=			s_ScriptFile ,								(*auszuführende Datei bat oder vbs eintragen*)
	i16_Timeout:= 	100);											(*in sec*)
END_PROGRAM

(* POU EPT Lib/Daten/FB_StartWinProcess, ST *)
FUNCTION_BLOCK FB_StartWinProcess
VAR_INPUT
	st_ctrl_in			:struct_ctrl_in;
	st_config			: struct_config;
	s_path				:STRING(255);		(*Pfad der Bat- oder vbs- Datei*)
	s_info_file			:STRING(255);		(*Pfad + Dateiname der Statusdatei*)
	s_script				:STRING;
	i16_Timeout			:INT;			(*in sec*)
	b_Start				:BOOL;
END_VAR
VAR_OUTPUT
	st_ctrl_out				:struct_ctrl_out;
	ErrId					:UDINT;
	ErrTyp					:STRING(5);
	ErrorMsg				:STRING(255);
	MsgString				:STRING(255);
END_VAR
VAR
	b_init					:BOOL;
	fb_state_entry			:ST_StateEntry;

	NT_StartProcess 		:NT_StartProcess;
	fbFileOpen				:FB_FileOpen;
	fbFileRead				:FB_FileRead;
	fbFileClose				:FB_FileClose;
	fbFileDelete				:FB_FileDelete;
	hFile					:UINT;

	fb_ton_wz				:TON;
	fb_ton_quitt				:TON;
	pos						:INT;
	FileString				:STRING(255);
	i16_Time				:INT;	(*in sec*)
	i						:INT;
	b_sm					:ARRAY[0..9] OF BOOL;	(*Störmeldungen aus der bat oder vbs Datei*)
	b_bm					:ARRAY[0..9] OF BOOL;	(*Bertiebsmeldungen aus der bat oder vbs Datei*)
	(*sonstige Meldungen*)
	sm_DateiNichtVorhanden				:BOOL;
	sm_FehlerBeimOeffnenDerDatei		:BOOL;
	sm_FehlerBeimAuslesenDerDatei		:BOOL;
	sm_FehlerBeimSchliessenDerDatei		:BOOL;
	sm_FehlerBeimLoeschenDerDatei		:BOOL;
	sm_KeineImportdateiVorhanden		:BOOL;
	sm_KeineErrIdGefunden				:BOOL;
END_VAR
(*======================================================
   FB: Start eines Win Prozess mit Prüfung 
 ------------------------------------------------------
   Auth: 		Werner Friedl   						 
   Date: 		19.02.2019   						     
   Rev.: 		1.0	
   Desc:		Eine Bat- oder vbs- Datei kann gestartet weden und der Status kommt über die ErrId wieder zurück.
			Die "ErrId" wird dann b_sm[ErrId] oder b_bm[ErrId], Damit können Betriebs und Störmeldungen von der bat angezeigt werden. 
			alle Meldungen quittieren sich selbst
			b_bm[0] =	'OK',
			b_sm[1] =	Netzwerk nicht verbunden!
			b_sm[2] =	User nicht vorhanden oder Passwort falsch!
			b_sm[3] =	Verzeichnis nicht vorhanden!
			b_sm[4] =	Datei nicht vorhanden!

   Historie:   1.0

   Aufruf Beispiel:
	s_instanz_name:='test',
	s_path:= 		s_tools_path,			(*Verzeichnis der Bat- und Prüf- Datei*)
	s_info_file:=	CONCAT(s_tools_path,'Test.txt') ,	(*Datei in der die Prüfung landet (sollte so heißen wie die Bat-Datei)*)
	s_script:=		'Test.bat' ,				(*auszuführende Datei bat oder vbs eintragen*)
	i16_Timeout:= 100);					(*in sec*)

 ========================================================*)
IF	NOT b_init THEN
	b_Init:=TRUE;
END_IF
(* ========================================================*)
fb_ton_quitt(IN:= , PT:= t#100ms, Q=> , ET=> );

fb_state_entry(i16_pos:= 1);
CASE fb_state_entry.i16_step OF
(*=======================================================*)
INIT_OBJ:
		fb_state_entry.i16_next_step := INIT;

(*=======================================================*)
INIT:	(*initialisieren*)
	IF fb_state_entry.E THEN
		fb_ton_quitt.IN := FALSE;
		st_ctrl_out.b_fehler := FALSE;
		st_ctrl_out.b_gestoppt := FALSE;
		st_ctrl_out.b_bereit := FALSE;
		st_ctrl_out.b_fertig := FALSE;
		st_ctrl_out.b_busy := FALSE;

		sm_DateiNichtVorhanden:=FALSE;
		sm_FehlerBeimOeffnenDerDatei:=FALSE;
		sm_FehlerBeimAuslesenDerDatei:=FALSE;
		sm_FehlerBeimSchliessenDerDatei:=FALSE;
		sm_FehlerBeimLoeschenDerDatei:=FALSE;
		sm_KeineImportdateiVorhanden:=FALSE;
		sm_KeineErrIdGefunden:=FALSE;
		FOR i:=0 TO 9 DO
			b_sm[i]:=FALSE;
			b_bm[i]:=FALSE;
		END_FOR
	END_IF

	(*-----------------------Weiterschaltbedingungen----------------------------*)
	fb_state_entry.i16_next_step:=BEREIT;

(*=======================================================*)
BEREIT: fb_state_entry.s_debugtext:='warte auf start';

	IF fb_state_entry.E THEN
		st_ctrl_out.b_bereit:=TRUE;
	END_IF

	(*-----------------------Weiterschaltbedingungen----------------------------*)
	IF	st_ctrl_in.b_start THEN
		NT_StartProcess.START:=TRUE;
		fb_state_entry.i16_next_step:=110;
	END_IF

	IF fb_state_entry.X THEN
		i16_Time:=0;
		st_ctrl_out.b_busy:=TRUE;
		st_ctrl_out.b_bereit := FALSE;
		st_ctrl_out.b_fertig := FALSE;
		ErrId:=99;
		ErrorMsg:='';
		FileString:='';
		MsgString:='';
	END_IF

	IF 	fb_state_entry.X THEN
		NT_StartProcess.START:=FALSE;
	END_IF

(*=======================================================*)
110:  fb_state_entry.s_debugtext:='start Datei öffnen';

	IF	fb_state_entry.fb_ton_Step.ET > t#1s THEN
		fbFileOpen.sPathName:=s_info_file;
   		fbFileOpen.bExecute:=TRUE;
	END_IF

	(*-----------------------Weiterschaltbedingungen----------------------------*)
	IF 	fbFileOpen.bBusy THEN
		fb_state_entry.i16_next_step:=120;
	END_IF

	IF 	fb_state_entry.X THEN
		ErrorMsg:='';
		st_ctrl_out.b_fehler:=FALSE;
	END_IF

(*=======================================================*)
120:  fb_state_entry.s_debugtext:='warte auf fertig Datei öffnen';

	IF 	NOT fbFileOpen.bBusy AND fb_state_entry.i16_next_step=120 THEN
		fbFileOpen.bExecute:=FALSE;
		IF	NOT fbFileOpen.bError THEN
			fb_state_entry.i16_next_step:=130;
		ELSIF
			fb_state_entry.fb_ton_Step.ET > t#1000ms THEN

			IF	i16_Time<=i16_Timeout THEN (*Datei nicht vorhanden*)
				fb_state_entry.i16_next_step:=110;
				i16_Time:=i16_Time+1;
			ELSE
				ErrId:=fbFileOpen.nErrId;
				fb_state_entry.i16_next_step:=FEHLER;

				IF 	fbFileOpen.nErrId =1804 THEN (*Datei nicht vorhanden*)
					sm_DateiNichtVorhanden:=TRUE;
					ErrorMsg:='Info Datei nicht vorhanden';
				ELSE
					sm_FehlerBeimOeffnenDerDatei:=TRUE;
					ErrorMsg:='Fehler beim Öffnen der Datei.';
				END_IF

			END_IF

		END_IF
	END_IF

(*=======================================================*)
130:  fb_state_entry.s_debugtext:='Start String aus Datei auslesen';

	fbFileRead.bExecute:=TRUE;
	IF 	fbFileRead.bBusy THEN
		fb_state_entry.i16_next_step:=140;
	END_IF

(*=======================================================*)
140:  fb_state_entry.s_debugtext:='warte auf fertig String aus Datei auslesen';

	IF 	NOT fbFileRead.bBusy THEN
		fbFileRead.bExecute:=FALSE;
		IF 	fbFileRead.bError THEN
			ErrId:=fbFileRead.nErrId;
			fb_state_entry.i16_next_step:=FEHLER;
			sm_FehlerBeimAuslesenDerDatei:=TRUE;
			ErrorMsg:='Fehler beim Auslesen der Datei.';
		ELSE
			fb_state_entry.i16_next_step:=150;
		END_IF
	END_IF

(*=======================================================*)
150: fb_state_entry.s_debugtext:='start Datei schließen';

	fbFileClose.bExecute:=TRUE;
	IF 	fbFileClose.bBusy THEN
		fb_state_entry.i16_next_step:=160;
	END_IF

(*=======================================================*)
160: fb_state_entry.s_debugtext:='warte auf fertig Datei schließen';

	IF 	NOT fbFileClose.bBusy THEN
		fbFileClose.bExecute:=FALSE;
		IF 	fbFileClose.bError THEN
			ErrId:=fbFileClose.nErrId;
			fb_state_entry.i16_next_step:=FEHLER;
			sm_FehlerBeimSchliessenDerDatei:=TRUE;
			ErrorMsg:='Fehler beim Schließen der Datei.';
		ELSE
			fb_state_entry.i16_next_step:=190;
		END_IF
	END_IF

(*=======================================================*)
170: fb_state_entry.s_debugtext:='start Datei löschen';

	fbFileDelete.bExecute:=TRUE;
	fbFileDelete.sPathName:=s_info_file;
	IF 	fbFileDelete.bBusy THEN
		fb_state_entry.i16_next_step:=180;
	END_IF

(*=======================================================*)
180: fb_state_entry.s_debugtext:='warte auf fertig Datei löschen';

	IF 	NOT fbFileDelete.bBusy THEN
		fbFileDelete.bExecute:=FALSE;
		IF 	fbFileDelete.bError THEN
			ErrId:=fbFileDelete.nErrId;
			fb_state_entry.i16_next_step:=FEHLER;
			sm_FehlerBeimLoeschenDerDatei:=TRUE;
			ErrorMsg:='Fehler beim löschen der Datei.';
		ELSE
			fb_state_entry.i16_next_step:=190;
		END_IF
	END_IF

(*=======================================================*)
190: fb_state_entry.s_debugtext:='Auswertung';

	IF 	fb_state_entry.E THEN
		MsgString:=FileString;

		(*falls noch ein Text mitkommt*)
		pos:=0;
		pos:=FIND (MsgString,'$N');
		IF 	pos >0 THEN
			ErrTyp:=LEFT(MsgString,pos-1);
			ErrId:=STRING_TO_INT(DELETE(ErrTyp,2,1));
			MsgString:=DELETE(MsgString,LEN(MsgString)-pos+2,pos);
		END_IF

		pos:=0;
		pos:=FIND (MSGString,'$T');
		IF 	pos >0 THEN
			MsgString:=DELETE(MsgString,1,pos);
		END_IF

	END_IF

	IF	LEN(FileString) = 0 THEN
		fb_state_entry.i16_next_step:=FEHLER;
		sm_KeineImportdateiVorhanden:=TRUE;
		ErrorMsg:='Kein Importstring vorhanden.';
	ELSE
		IF	ErrId <>99 THEN
			IF	FIND(ErrTyp,'BM') > 0 THEN
				b_bm[ErrId]:=TRUE;
			ELSIF	FIND(ErrTyp,'SM') > 0 THEN
				b_sm[ErrId]:=TRUE;
			END_IF
			fb_state_entry.i16_next_step:=200;
		ELSE
			sm_KeineErrIdGefunden:=TRUE;
			ErrorMsg:='**Error Id not found**';
			fb_state_entry.i16_next_step:=FEHLER;
		END_IF
	END_IF

(*=======================================================*)
200: fb_state_entry.s_debugtext:='Fertig';

	IF	fb_state_entry.fb_ton_Step.ET >t#5s THEN
		IF	FIND(ErrTyp,'BM') > 0 THEN
			fb_state_entry.i16_next_step:=INIT;
			st_ctrl_out.b_fertig:=TRUE;
		ELSE
			fb_state_entry.i16_next_step:=FEHLER;
		END_IF

	END_IF

	IF fb_state_entry.X THEN
		st_ctrl_out.b_busy:=FALSE;
	END_IF

(*=======================================================*)
STOP, FEHLER:

	IF fb_state_entry.E THEN
		st_ctrl_out.b_fehler := fb_state_entry.i16_step = FEHLER;
		st_ctrl_out.b_gestoppt := fb_state_entry.i16_step = STOP;
		st_ctrl_out.b_busy:=FALSE;
		fb_ton_wz.IN:=TRUE;
	END_IF

	IF	fb_state_entry.fb_ton_Step.ET >t#5s THEN   (*Quittiert sich selbst*)
		fb_state_entry.i16_next_step:=INIT;
	END_IF

	IF fb_state_entry.X THEN
		fb_ton_wz.IN:=FALSE;
	END_IF

END_CASE
(*=======================================================*)
fb_state_entry(i16_pos:= 2);
st_ctrl_in:=st_ctrl_in_empty;

(* Fehlermeldungen und Betriebsmeldungen ab dem Startindex in die Meldungsarrays des fb_Fehlermeldung schreiben *)
garr_stoermeldungen[st_config.i16_meld_startindex +0] := b_sm[0];
garr_stoermeldungen[st_config.i16_meld_startindex +1] := b_sm[1];		(*Netzwerk nicht verbunden*)
garr_stoermeldungen[st_config.i16_meld_startindex +2] := b_sm[2];		(*User nicht vorhanden oder Passwort falsch*)
garr_stoermeldungen[st_config.i16_meld_startindex +3] := b_sm[3];		(*Verzeichnis nicht vorhanden!*)
garr_stoermeldungen[st_config.i16_meld_startindex +4] := b_sm[4];		(*Datei nicht vorhanden!*)
garr_stoermeldungen[st_config.i16_meld_startindex +5] := b_sm[5];
garr_stoermeldungen[st_config.i16_meld_startindex +6] := b_sm[6];
garr_stoermeldungen[st_config.i16_meld_startindex +7] := b_sm[7];
garr_stoermeldungen[st_config.i16_meld_startindex +8] := b_sm[8];
garr_stoermeldungen[st_config.i16_meld_startindex +9] := b_sm[9];
garr_stoermeldungen[st_config.i16_meld_startindex +10] := sm_DateiNichtVorhanden;
garr_stoermeldungen[st_config.i16_meld_startindex +11] := sm_FehlerBeimOeffnenDerDatei;
garr_stoermeldungen[st_config.i16_meld_startindex +12] := sm_FehlerBeimAuslesenDerDatei;
garr_stoermeldungen[st_config.i16_meld_startindex +13] := sm_FehlerBeimSchliessenDerDatei;
garr_stoermeldungen[st_config.i16_meld_startindex +14] := sm_FehlerBeimLoeschenDerDatei;
garr_stoermeldungen[st_config.i16_meld_startindex +15] := sm_KeineImportdateiVorhanden;
garr_stoermeldungen[st_config.i16_meld_startindex +16] := sm_KeineErrIdGefunden;
garr_stoermeldungen[st_config.i16_meld_startindex +17] := FALSE;
garr_stoermeldungen[st_config.i16_meld_startindex +18] := FALSE;
garr_stoermeldungen[st_config.i16_meld_startindex +19] := FALSE;

garr_betriebsmeldungen[st_config.i16_meld_startindex + 0] := b_bm[0];		(*OK*)
garr_betriebsmeldungen[st_config.i16_meld_startindex + 1] := b_bm[1];		(*keinen Unterschied gefunden*)
garr_betriebsmeldungen[st_config.i16_meld_startindex + 2] := b_bm[2];
garr_betriebsmeldungen[st_config.i16_meld_startindex + 3] := b_bm[3];
garr_betriebsmeldungen[st_config.i16_meld_startindex + 4] := b_bm[4];
garr_betriebsmeldungen[st_config.i16_meld_startindex + 5] := b_bm[5];
garr_betriebsmeldungen[st_config.i16_meld_startindex + 6] := b_bm[6];
garr_betriebsmeldungen[st_config.i16_meld_startindex + 7] := b_bm[7];
garr_betriebsmeldungen[st_config.i16_meld_startindex + 8] := b_bm[8];
garr_betriebsmeldungen[st_config.i16_meld_startindex + 9] := b_bm[9];


CallPrg();
END_FUNCTION_BLOCK
ACTION CallPrg:
IF 	FIND(s_script,'.bat') > 0 THEN


	NT_StartProcess(
		NETID:='',
		PATHSTR		:='C:\Windows\System32\cmd.exe',
		DIRNAME		:=s_path,
		COMNDLINE	:=CONCAT('/C start /b ', s_script),
		START			:=,
		TMOUT			:=DEFAULT_ADS_TIMEOUT);

ELSE
	NT_StartProcess(
		NETID:='',
		PATHSTR	:='C:\Windows\System32\wscript.exe',
		DIRNAME	:=s_path,
		COMNDLINE	:=s_script,
		START		:=,
		TMOUT		:=DEFAULT_ADS_TIMEOUT);
END_IF

fbFileOpen(
	sNetId:='',
	sPathName:= ,
	nMode:=FOPEN_MODEREAD,
	ePath:=PATH_GENERIC,
	bExecute:= ,
	tTimeout:=T#1s,
	hFile=> hFile);

fbFileRead(
	sNetId:='' ,
	hFile:=hFile,
	pReadBuff:= ADR(FileString)  ,
	cbReadLen:=SIZEOF(FileString)  ,
	tTimeout:=t#2s );

fbFileClose(
	sNetId:='',
	hFile:=hFile,
	bExecute:= ,
	tTimeout:=t#1s);

fbFileDelete(
	sNetId:= ,
	sPathName:= , 
	ePath:= PATH_GENERIC,
	bExecute:= ,
	tTimeout:= t#1s );
END_ACTION

(* POU EPT Lib/Daten/ST_SaveAndLoad, ST *)
PROGRAM ST_SaveAndLoad
VAR_INPUT
	st_ctrl_in			: struct_ctrl_in;
	st_config			: struct_config;

END_VAR
VAR_OUTPUT
	st_ctrl_out			:struct_ctrl_out;
END_VAR
VAR
	b_init				:BOOL;
	fb_state_entry		:ST_StateEntry;
	fb_ton_quitt			:TON;

	NT_StartProcess 	: NT_StartProcess;
	fbFileDelete			: FB_FileDelete;

	s_script				: STRING;
	sm_FehlerBeimStartenDerBat				:BOOL;
	sm_FehlerBeimLoeschenDerDatei		:BOOL;

END_VAR
VAR CONSTANT
		s_bbgenMachineToSrv				:STRING:=		'_bbgen_aktuelles_wz_und_band_von_zelle_nach_server.bat';

		s_bbgenSrvToMachine				:STRING:=		'_bbgen_von_server_nach_zelle.bat';
		s_bbgenSrvToMachineHalbauto		:STRING:=		'_bbgen_von_server_nach_zelle_halbauto.bat';
		s_bbgenSrvToMachineManuell		:STRING:=		'_bbgen_von_server_nach_zelle_manuell.bat';

		s_fbwf_info							:STRING:=		'fbwf_info.bat';
		s_fbwf_disable						:STRING:=		'fbwf_disable.bat';
		s_fbwf_enable						:STRING:=		'fbwf_enable.bat';
END_VAR
(*======================================================
   ST_SaveAndLoad
 ------------------------------------------------------
   Auth: 		Werner Friedl   						 
   Date: 		06.10.2020   						     
   Rev.: 		1.0	
   Desc:		Die bat Datein zum laden und speichern der BBgen Dateien werden hier ausgeführt.
			mit der Constante b_wkzBereinigen kann bestimmt werden, ob die Werkzeugdateu forher gelöscht wird.

 ========================================================*)
IF	NOT b_init THEN
	b_Init:=TRUE;
END_IF
CallPrg();
(* ========================================================*)
fb_ton_quitt(IN:= , PT:= t#100ms, Q=> , ET=> );



fb_state_entry(i16_pos:= 1);
CASE fb_state_entry.i16_step OF
(*=======================================================*)
INIT_OBJ:
		fb_state_entry.i16_next_step := INIT;

(*=======================================================*)
INIT:
	IF	fb_state_entry.E THEN
		sm_FehlerBeimStartenDerBat:=FALSE;
		sm_FehlerBeimLoeschenDerDatei:=FALSE;
	END_IF

		fb_state_entry.i16_next_step := BEREIT;


(*=======================================================*)
BEREIT:	fb_state_entry.s_debugtext:='warte auf Taster Save oder Load';

	IF fb_state_entry.E THEN
		st_ctrl_out.b_bereit:=TRUE;
		NT_StartProcess.START:=FALSE;
	END_IF

	(*-----------------------Weiterschaltbedingungen----------------------------*)
	IF 	visu.b_load THEN
		fb_state_entry.i16_next_step:=110;
	ELSIF
		visu.b_save THEN
		IF 	gst_datensatz.st_md.b_wkzBereinigen THEN
			fb_state_entry.i16_next_step:=210;
		ELSE
			fb_state_entry.i16_next_step:=240;
		END_IF
	ELSIF
		visu.b_fbwf_info THEN
		s_script:=s_fbwf_info;
		fb_state_entry.i16_next_step:=120;
	ELSIF
		visu.b_fbwf_disable THEN
		s_script:=s_fbwf_disable;
		fb_state_entry.i16_next_step:=120;
	ELSIF
		visu.b_fbwf_enable THEN
		s_script:=s_fbwf_enable;
		fb_state_entry.i16_next_step:=120;
	END_IF

	IF fb_state_entry.X THEN
		st_ctrl_out.b_busy:=TRUE;
		st_ctrl_out.b_bereit := FALSE;
		st_ctrl_out.b_fertig := FALSE;
	END_IF

(*=======================================================*)
110:fb_state_entry.s_debugtext:='erstelle s_script';

	IF fb_state_entry.E THEN

 		CASE gst_datensatz.st_md.i16_typ_bestueckmodus OF

			BESTUECKUNG_MANUAL:
				s_script:=CONCAT(visu.s_akt_sprache,s_bbgenSrvToMachineManuell);

			BESTUECKUNG_HALBAUTO:
				s_script:=CONCAT(visu.s_akt_sprache,s_bbgenSrvToMachineHalbauto);

			BESTUECKUNG_AUTO:
				s_script:=CONCAT(visu.s_akt_sprache,s_bbgenSrvToMachine);
		END_CASE

		fb_state_entry.i16_next_step:=120;
	END_IF

(*=======================================================*)
120:fb_state_entry.s_debugtext:='start bat Script "Laden der Dateien vom Server"';

	IF 	fb_state_entry.E THEN
		NT_StartProcess.START:=TRUE;
	END_IF

	(*-----------------------Weiterschaltbedingungen----------------------------*)
	IF 	NT_StartProcess.BUSY THEN
		fb_state_entry.i16_next_step:=130;
	END_IF

	IF 	fb_state_entry.X THEN
		NT_StartProcess.START:=FALSE;
	END_IF

(*=======================================================*)
130:fb_state_entry.s_debugtext:='Warten auf fertig';

	IF 	NT_StartProcess.ERR THEN
		fb_state_entry.s_debugtext:=CONCAT(fb_state_entry.s_debugtext,' ERRID => ');
		fb_state_entry.s_debugtext:=CONCAT(fb_state_entry.s_debugtext,UDINT_TO_STRING(NT_StartProcess.ERRID));
		sm_FehlerBeimStartenDerBat:=TRUE;
		fb_state_entry.i16_next_step:=FEHLER;
	ELSIF
		NOT NT_StartProcess.BUSY AND
		NOT NT_StartProcess.ERR AND
		fb_state_entry.fb_ton_Step.ET>t#3000ms THEN
		st_ctrl_out.b_busy:=FALSE;
		st_ctrl_out.b_fertig := TRUE;
		fb_state_entry.i16_next_step:=BEREIT;
	END_IF

	IF 	fb_state_entry.X THEN
		visu.b_fbwf_info:=FALSE;
		visu.b_fbwf_disable:=FALSE;
		visu.b_fbwf_enable:=FALSE;
		visu.b_load:=FALSE;
	END_IF

(*=======================================================*)
(*=======================================================*)
210:	fb_state_entry.s_debugtext:='Löschen der Werkzeug Datei';

	IF 	fb_state_entry.E THEN
		fbFileDelete.sPathName:=CONCAT(CONCAT(ST_BBGen.s_wkz_path,gst_datensatz.st_md.s_aktuelles_wkz),'.xml');
		fbFileDelete.bExecute:=TRUE;
	END_IF

	(*-----------------------Weiterschaltbedingungen----------------------------*)
	IF 	fbFileDelete.bBusy THEN
		fb_state_entry.i16_next_step:=220;
	END_IF

	IF 	fb_state_entry.X THEN
		fbFileDelete.bExecute:=FALSE;
	END_IF

(*=======================================================*)
220: fb_state_entry.s_debugtext:='warte auf fertig';

	IF 	NOT fbFileDelete.bBusy THEN
		IF 	fbFileDelete.bError THEN
			fb_state_entry.s_debugtext:=CONCAT(fb_state_entry.s_debugtext,' ERRID => ');
			fb_state_entry.s_debugtext:=CONCAT(fb_state_entry.s_debugtext,UDINT_TO_STRING(fbFileDelete.nErrId));
			fb_state_entry.i16_next_step:=FEHLER;
			sm_FehlerBeimLoeschenDerDatei:=TRUE;
		ELSE
			fb_state_entry.i16_next_step:=230;
		END_IF
	END_IF

(*=======================================================*)
230: fb_state_entry.s_debugtext:='Werkzeugdatei neu erstellen';

	IF 	fb_state_entry.E THEN
		gi16_bbgen_auftrag:=SCHREIBE_WKZ;
	END_IF

	(*-----------------------Weiterschaltbedingungen----------------------------*)
	IF 	gi16_bbgen_auftrag = KEIN_BB_AUFTRAG THEN
		fb_state_entry.i16_next_step:=240;
	END_IF

(*=======================================================*)
240:	fb_state_entry.s_debugtext:='Speichern auf Server';

	IF 	fb_state_entry.E THEN
		s_script:=CONCAT(visu.s_akt_sprache,s_bbgenMachineToSrv);
		NT_StartProcess.START:=TRUE;
	END_IF

	(*-----------------------Weiterschaltbedingungen----------------------------*)
	IF 	NT_StartProcess.BUSY THEN
		fb_state_entry.i16_next_step:=250;
	END_IF

	IF 	fb_state_entry.X THEN
		NT_StartProcess.START:=FALSE;
	END_IF

(*=======================================================*)
250:fb_state_entry.s_debugtext:='Warten auf fertig';

	IF 	NT_StartProcess.ERR THEN
		fb_state_entry.s_debugtext:=CONCAT(fb_state_entry.s_debugtext,' ERRID => ');
		fb_state_entry.s_debugtext:=CONCAT(fb_state_entry.s_debugtext,UDINT_TO_STRING(NT_StartProcess.ERRID));
		sm_FehlerBeimStartenDerBat:=TRUE;
		fb_state_entry.i16_next_step:=FEHLER;
	ELSIF
		NOT NT_StartProcess.BUSY AND
		NOT NT_StartProcess.ERR AND
		fb_state_entry.fb_ton_Step.ET>t#3000ms THEN
		st_ctrl_out.b_busy:=FALSE;
		st_ctrl_out.b_fertig := TRUE;
		fb_state_entry.i16_next_step:=BEREIT;
	END_IF

	IF 	fb_state_entry.X THEN
		visu.b_save:=FALSE;
	END_IF

(*=======================================================*)
STOP, FEHLER:

	IF fb_state_entry.E THEN
		st_ctrl_out.b_fehler := fb_state_entry.i16_step = FEHLER;
		st_ctrl_out.b_gestoppt := fb_state_entry.i16_step = STOP;
		st_ctrl_out.b_busy:=FALSE;
	END_IF

	IF	fb_state_entry.fb_ton_Step.ET > t#1000ms THEN   (*Quittiert sich selbst*)
		fb_state_entry.i16_next_step:=INIT;
	END_IF

END_CASE

fb_state_entry(i16_pos:= 2 );
st_ctrl_in:=st_ctrl_in_empty;


garr_stoermeldungen[st_config.i16_meld_startindex + 0] := sm_FehlerBeimStartenDerBat;
garr_stoermeldungen[st_config.i16_meld_startindex + 1] := sm_FehlerBeimLoeschenDerDatei;
garr_stoermeldungen[st_config.i16_meld_startindex + 2] := FALSE;
garr_stoermeldungen[st_config.i16_meld_startindex + 3] := FALSE;
garr_stoermeldungen[st_config.i16_meld_startindex + 4] := FALSE;
garr_stoermeldungen[st_config.i16_meld_startindex + 5] := FALSE;
garr_stoermeldungen[st_config.i16_meld_startindex + 6] := FALSE;
garr_stoermeldungen[st_config.i16_meld_startindex + 7] := FALSE;
garr_stoermeldungen[st_config.i16_meld_startindex + 8] := FALSE;
garr_stoermeldungen[st_config.i16_meld_startindex + 9] := FALSE;
garr_stoermeldungen[st_config.i16_meld_startindex + 10] := FALSE;
garr_stoermeldungen[st_config.i16_meld_startindex + 11] := FALSE;
garr_stoermeldungen[st_config.i16_meld_startindex + 12] := FALSE;
garr_stoermeldungen[st_config.i16_meld_startindex + 13] := FALSE;
garr_stoermeldungen[st_config.i16_meld_startindex + 14] := FALSE;
garr_stoermeldungen[st_config.i16_meld_startindex + 15] := FALSE;
garr_stoermeldungen[st_config.i16_meld_startindex + 16] := FALSE;
garr_stoermeldungen[st_config.i16_meld_startindex + 17] := FALSE;
garr_stoermeldungen[st_config.i16_meld_startindex + 18] := FALSE;
garr_stoermeldungen[st_config.i16_meld_startindex + 19] := FALSE;

garr_betriebsmeldungen[st_config.i16_meld_startindex + 0] := FALSE;
garr_betriebsmeldungen[st_config.i16_meld_startindex + 1] := FALSE;
garr_betriebsmeldungen[st_config.i16_meld_startindex + 2] := FALSE;
garr_betriebsmeldungen[st_config.i16_meld_startindex + 3] := FALSE;
garr_betriebsmeldungen[st_config.i16_meld_startindex + 4] := FALSE;
garr_betriebsmeldungen[st_config.i16_meld_startindex + 5] := FALSE;
garr_betriebsmeldungen[st_config.i16_meld_startindex + 6] := FALSE;
garr_betriebsmeldungen[st_config.i16_meld_startindex + 7] := FALSE;
garr_betriebsmeldungen[st_config.i16_meld_startindex + 8] := FALSE;
garr_betriebsmeldungen[st_config.i16_meld_startindex + 9] := FALSE;
garr_betriebsmeldungen[st_config.i16_meld_startindex + 10] := FALSE;
garr_betriebsmeldungen[st_config.i16_meld_startindex + 11] := FALSE;
garr_betriebsmeldungen[st_config.i16_meld_startindex + 12] := FALSE;
garr_betriebsmeldungen[st_config.i16_meld_startindex + 13] := FALSE;
garr_betriebsmeldungen[st_config.i16_meld_startindex + 14] := FALSE;
garr_betriebsmeldungen[st_config.i16_meld_startindex + 15] := FALSE;
garr_betriebsmeldungen[st_config.i16_meld_startindex + 16] := FALSE;
garr_betriebsmeldungen[st_config.i16_meld_startindex + 17] := FALSE;
garr_betriebsmeldungen[st_config.i16_meld_startindex + 18] := FALSE;
garr_betriebsmeldungen[st_config.i16_meld_startindex + 19] := FALSE;
END_PROGRAM
ACTION CallPrg:
NT_StartProcess(
	NETID:='',
	PATHSTR		:='C:\Windows\System32\cmd.exe',
	DIRNAME		:=s_tools_path,
	COMNDLINE	:=CONCAT('/C start /b ', s_script),
	START			:=,
	TMOUT			:=DEFAULT_ADS_TIMEOUT);


fbFileDelete(
	sNetId:= ,
	sPathName:= , 
	ePath:= PATH_GENERIC,
	bExecute:= ,
	tTimeout:= t#1s );
END_ACTION

(* POU Gemeinsamkeiten17xx/Initialisierung/Startup/ST_Datainit_Stationen, ST *)
PROGRAM ST_Datainit_Stationen
VAR
	b_config_fertig			: BOOL := FALSE;
	i						: INT := 0;
	Index					: INT := 0;
END_VAR
IF	NOT betriebsarten.st_config.b_config_fertig OR
	NOT betriebsfreigaben.st_config.b_config_fertig OR
	NOT stoerungen_quittieren.st_config.b_config_fertig OR
	NOT bandeinzug_kontroller.st_config.b_config_fertig OR
	NOT wt_transport_kontroller.st_config.b_config_fertig OR
	NOT wt_transport_beladen.st_config.b_config_fertig OR
	NOT wt_transport_abgabe.st_config.b_config_fertig OR
	NOT routing_backpanel.st_config.b_config_fertig OR
	NOT routing_nachbarpc.st_config.b_config_fertig OR
	NOT UPS.st_config.b_config_fertig OR
	NOT haspel_kontroller.st_config.b_config_fertig OR
	NOT haspel_li.fb.st_config.b_config_fertig OR
	NOT haspel_re.fb.st_config.b_config_fertig OR
	NOT hublift_links.st_config.b_config_fertig OR
	NOT hublift_rechts.st_config.b_config_fertig OR
	NOT wkz_absicherung.st_config.b_config_fertig OR
	NOT stueckzahlen.fb.st_config.b_config_fertig OR
	NOT bandwechsel_kontroller.st_config.b_config_fertig OR
	NOT bandspruehoeler.st_config.b_config_fertig OR
	NOT einpresskraft_kontroller.st_config.b_config_fertig OR
	NOT kraftmessdose.fb.st_config.b_config_fertig OR
	NOT nockenschaltwerk_bestueckachse.st_config.b_config_fertig OR
	NOT safety.st_config.b_config_fertig OR
	NOT xml_server.st_config.b_config_fertig OR
	NOT fb_edit_mfps_bestuecken_z.st_config.b_config_fertig OR
	NOT fb_edit_mfps_bestuecken_y.st_config.b_config_fertig OR
	NOT fb_edit_mfps_yz_tisch.st_config.b_config_fertig OR
	NOT fb_camtable_bestueckachse.st_config.b_config_fertig OR
	NOT fb_edit_mfps_bestuecken_b.st_config.b_config_fertig OR
	NOT bbgen.st_config.b_config_fertig OR
	NOT barcode.fb.st_config.b_config_fertig OR
	NOT balluff_tag_reader.fb.st_config.b_config_fertig OR
	NOT wt_transport_warteposition_1720.st_config.b_config_fertig OR
	NOT wt_transport_beladen_1720.st_config.b_config_fertig OR
	NOT rasterfolienmontage.st_config.b_config_fertig OR
	NOT rasterfolieneinzug.st_config.b_config_fertig OR
	NOT Lesen_Schreiben_Tag.st_config.b_config_fertig OR
	NOT Service.st_config.b_config_fertig OR
	NOT ST_TouchProbe.st_config.b_config_fertig OR
	NOT wt_transport_warteposition_1700.st_config.b_config_fertig OR
	NOT wt_transport_beladen_achse_1700.st_config.b_config_fertig OR
	NOT EtherCatDiag[1].st_config.b_config_fertig
	THEN
		(* Betriebsarten *)
		betriebsarten.st_config.b_config_fertig := FALSE;
		betriebsarten.st_config.b_station_aktiv := TRUE;
		betriebsarten.st_config.i16_meld_startindex := 20;
		betriebsarten.st_config.str_beschreibung := ' ';
		betriebsarten.st_config.str_instanz_name := 'Betriebsarten';
		betriebsarten.st_config.b_config_fertig := TRUE;
		
		(* Betriebsfreigaben *)
		betriebsfreigaben.st_config.b_config_fertig := FALSE;
		betriebsfreigaben.st_config.b_station_aktiv := TRUE;
		betriebsfreigaben.st_config.i16_meld_startindex := 40;
		betriebsfreigaben.st_config.str_beschreibung := ' ';
		betriebsfreigaben.st_config.str_instanz_name := 'Betriebsfeigaben';
		betriebsfreigaben.st_config.b_config_fertig := TRUE;
		
		(* Störungen quittieren *)
		stoerungen_quittieren.st_config.b_config_fertig := FALSE;
		stoerungen_quittieren.st_config.b_station_aktiv := TRUE;
		stoerungen_quittieren.st_config.i16_meld_startindex := 60;
		stoerungen_quittieren.st_config.str_beschreibung := ' ';
		stoerungen_quittieren.st_config.str_instanz_name := 'Störungen quittieren';
		stoerungen_quittieren.st_config.b_config_fertig := TRUE;

		(* Bandeinzugskontroller *)
		bandeinzug_kontroller.st_config.b_config_fertig := FALSE;
		bandeinzug_kontroller.st_config.b_station_aktiv := TRUE;
		bandeinzug_kontroller.st_config.i16_meld_startindex := 80;
		bandeinzug_kontroller.st_config.str_beschreibung := ' ';
		bandeinzug_kontroller.st_config.str_instanz_name := 'Bandeinzugkontroller';
		bandeinzug_kontroller.st_config.b_config_fertig := TRUE;
		
		(* WT-Transport Kontroller *)
		wt_transport_kontroller.st_config.b_config_fertig := FALSE;
		wt_transport_kontroller.st_config.i16_meld_startindex := 100;
		wt_transport_kontroller.st_config.str_beschreibung := ' ';
		wt_transport_kontroller.st_config.str_instanz_name := 'WT-Transport Kontroller';
		wt_transport_kontroller.st_config.b_config_fertig := TRUE;
		
		(* WT-Transport Beladestation*)
		wt_transport_beladen.st_config.b_config_fertig := FALSE;
		wt_transport_beladen.st_config.i16_meld_startindex := 120;
		wt_transport_beladen.st_config.str_beschreibung := ' ';
		wt_transport_beladen.st_config.str_instanz_name := 'WT-Transport Beladestation';
		wt_transport_beladen.st_config.b_config_fertig := TRUE;
		
		(* WT-Transport Abgabestation *)
		wt_transport_abgabe.st_config.b_config_fertig := FALSE;
		wt_transport_abgabe.st_config.i16_meld_startindex := 140;
		wt_transport_abgabe.st_config.str_beschreibung := ' ';
		wt_transport_abgabe.st_config.str_instanz_name := 'WT-Transport Abgabestation';
		wt_transport_abgabe.st_config.b_config_fertig := TRUE;
		
		(* Routing Backpanel *)
		routing_backpanel.st_config.b_config_fertig := FALSE;
		routing_backpanel.st_config.i16_meld_startindex := 160;
		routing_backpanel.st_config.str_beschreibung := ' ';
		routing_backpanel.st_config.str_instanz_name := 'Routing Backpanel';
		routing_backpanel.st_config.b_config_fertig := TRUE;
		
		(* Routing Nachbar-PCs *)
		routing_nachbarpc.st_config.b_config_fertig := FALSE;
		routing_nachbarpc.st_config.i16_meld_startindex := 180;
		routing_nachbarpc.st_config.str_beschreibung := ' ';
		routing_nachbarpc.st_config.str_instanz_name := 'Routing Nachbar-PCs';
		routing_nachbarpc.st_config.b_config_fertig := TRUE;
		
		(* Haspelkontroller *)
		haspel_kontroller.st_config.b_config_fertig := FALSE;
		haspel_kontroller.st_config.b_station_aktiv := TRUE;
		haspel_kontroller.st_config.i16_meld_startindex := 200;
		haspel_kontroller.st_config.str_beschreibung := ' ';
		haspel_kontroller.st_config.str_instanz_name := 'Haspelkontroller';
		haspel_kontroller.t_abschaltzeit_motor := t#60s;
		haspel_kontroller.b_drehrichtung_antrieb_links := FALSE;
		haspel_kontroller.st_config.b_config_fertig := TRUE;

		(* Haspel links *)
		haspel_li.fb.st_config.b_config_fertig := FALSE;
		haspel_li.fb.st_config.b_station_aktiv := TRUE;
		haspel_li.fb.st_config.i16_meld_startindex := 220;
		haspel_li.fb.st_config.str_beschreibung := ' ';
		haspel_li.fb.st_config.str_instanz_name := 'Haspel links';
		haspel_li.fb.t_wartezeit_bandende := t#2s;
		haspel_li.fb.st_config.b_config_fertig := TRUE;
		
		(* Haspel rechts *)
		haspel_re.fb.st_config.b_config_fertig := FALSE;
		haspel_re.fb.st_config.b_station_aktiv := TRUE;
		haspel_re.fb.st_config.i16_meld_startindex := 240;
		haspel_re.fb.st_config.str_beschreibung := ' ';
		haspel_re.fb.st_config.str_instanz_name := 'Haspel rechts';
		haspel_re.fb.t_wartezeit_bandende := t#2s;
		haspel_re.fb.st_config.b_config_fertig := TRUE;
		
		(* Hublift links *)
		hublift_links.st_config.b_config_fertig := FALSE;
		hublift_links.st_config.i16_meld_startindex := 280;
		hublift_links.st_config.str_beschreibung := ' ';
		hublift_links.st_config.str_instanz_name := 'Hublift links';
		hublift_links.st_config.b_config_fertig := TRUE;
		
		(* Hublift rechts *)
		hublift_rechts.st_config.b_config_fertig := FALSE;
		hublift_rechts.st_config.i16_meld_startindex := 300;
		hublift_rechts.st_config.str_beschreibung := ' ';
		hublift_rechts.st_config.str_instanz_name := 'Hublift rechts';
		hublift_rechts.st_config.b_config_fertig := TRUE;
		
		(* Werkzeugabsicherung *)
		wkz_absicherung.st_config.b_config_fertig := FALSE;
		wkz_absicherung.st_config.b_station_aktiv := TRUE;
		wkz_absicherung.st_config.i16_meld_startindex := 320;
		wkz_absicherung.st_config.str_beschreibung := ' ';
		wkz_absicherung.st_config.str_instanz_name := 'Werkzeugabsicherung';
		wkz_absicherung.st_config.b_config_fertig := TRUE;
		
		(* Stückzahlen *)
		stueckzahlen.fb.st_config.b_config_fertig := FALSE;
		stueckzahlen.fb.st_config.b_station_aktiv := TRUE;
		stueckzahlen.fb.st_config.i16_meld_startindex := 340;
		stueckzahlen.fb.st_config.str_beschreibung := ' ';
		stueckzahlen.fb.st_config.str_instanz_name := 'Stueckzahlen';
		stueckzahlen.fb.st_config.b_config_fertig := TRUE;
		
		(* Bandwechselkontroller *)
		bandwechsel_kontroller.st_config.b_config_fertig := FALSE;
		bandwechsel_kontroller.st_config.b_station_aktiv := TRUE;
		bandwechsel_kontroller.st_config.i16_meld_startindex := 360;
		bandwechsel_kontroller.st_config.str_beschreibung := ' ';
		bandwechsel_kontroller.st_config.str_instanz_name := 'Bandwechselkontroller';
		bandwechsel_kontroller.st_config.b_config_fertig := TRUE;
		
		(* Bandsprühöler *)
		bandspruehoeler.st_config.b_config_fertig := FALSE;
		bandspruehoeler.st_config.b_station_aktiv := TRUE;
		bandspruehoeler.st_config.i16_meld_startindex := 380;
		bandspruehoeler.st_config.str_beschreibung := ' ';
		bandspruehoeler.st_config.str_instanz_name := 'Bandsprühöler';
		bandspruehoeler.st_config.b_config_fertig := TRUE;

		(* UPS Überwachung *)
		UPS.st_config.b_config_fertig := FALSE;
		UPS.st_config.b_station_aktiv := TRUE;
		UPS.st_config.i16_meld_startindex := 440;		(*-445*)
		UPS.st_config.str_beschreibung := ' ';
		UPS.st_config.str_instanz_name := 'UPS Überwachung';
		UPS.st_config.b_config_fertig := TRUE;

		(*Einpresskraftkontroller *)
		einpresskraft_kontroller.st_config.b_config_fertig := FALSE;
		einpresskraft_kontroller.st_config.b_station_aktiv := TRUE;
		einpresskraft_kontroller.st_config.i16_meld_startindex := 460;
		einpresskraft_kontroller.st_config.str_beschreibung := ' ';
		einpresskraft_kontroller.st_config.str_instanz_name := 'Einpresskraftkontroller';

		CASE gst_datensatz.st_md.i16_typ_zelle OF
			KEINE_ZELLE:
				gst_datensatz.st_band.st_einpressen.st_einstellungen.enu_modus := KEIN_MODUS;
			BESTUECKZELLE_1700:
				gst_datensatz.st_band.st_einpressen.st_einstellungen.enu_modus := F_MAXWERT;
			BESTUECKZELLE_1720:
				gst_datensatz.st_band.st_einpressen.st_einstellungen.enu_modus := F_MAXWERT;
			RASTERFOLIE:
				gst_datensatz.st_band.st_einpressen.st_einstellungen.enu_modus := KEIN_MODUS;
		END_CASE

		einpresskraft_kontroller.st_config.b_config_fertig := TRUE;
		
		(* Kraftmessdose Kanal 1*)
		kraftmessdose.fb.st_config.b_config_fertig := FALSE;
		kraftmessdose.fb.st_config.b_station_aktiv := TRUE;
		kraftmessdose.fb.st_config.i16_meld_startindex := 480;
		kraftmessdose.fb.st_config.str_beschreibung := ' ';
		kraftmessdose.fb.st_config.str_instanz_name := 'Kraftmessdose Kanal 1';
		kraftmessdose.fb.st_config.b_config_fertig := TRUE;
		
		(* Nockenschaltwerk Bestückachse *)
		nockenschaltwerk_bestueckachse.st_config.b_config_fertig := FALSE;
		nockenschaltwerk_bestueckachse.st_config.b_station_aktiv := TRUE;
		nockenschaltwerk_bestueckachse.st_config.i16_meld_startindex := 500;
		nockenschaltwerk_bestueckachse.st_config.str_beschreibung := ' ';
		nockenschaltwerk_bestueckachse.st_config.str_instanz_name := 'Nockenschaltwerk Bestückachse';
		nockenschaltwerk_bestueckachse.st_config.b_config_fertig := TRUE;
		
		(* Nockenschaltwerk Z-Achse *)
		(* 520 *)
		
		(* Nockenschaltwerk Y-Achse *)
		(* 540 *)
		
		(* Frei *)
		(* 560 *)

		(* Safety *)
		safety.st_config.b_config_fertig := FALSE;
		safety.st_config.b_station_aktiv := TRUE;
		safety.st_config.i16_meld_startindex := 580;
		safety.st_config.str_beschreibung := ' ';
		safety.st_config.str_instanz_name := 'Safety';
		safety.st_config.b_config_fertig := TRUE;
		
		(* XML-Server *)
		xml_server.st_config.b_config_fertig := FALSE;
		xml_server.st_config.b_station_aktiv := TRUE;
		xml_server.st_config.i16_meld_startindex := 620;
		xml_server.st_config.str_beschreibung := ' ';
		xml_server.st_config.str_instanz_name := 'XML-Server';
		xml_server.st_config.b_config_fertig := TRUE;

		(* Kurvenscheibeneditor *)
		fb_edit_mfps_bestuecken_z.st_config.b_config_fertig := FALSE;
		fb_edit_mfps_bestuecken_z.st_config.b_station_aktiv := TRUE;
		fb_edit_mfps_bestuecken_z.st_config.i16_meld_startindex := 640;
		fb_edit_mfps_bestuecken_z.st_config.str_beschreibung := ' ';
		fb_edit_mfps_bestuecken_z.st_config.str_instanz_name := 'Kurvenscheibeneditor Bestücken Z-Achse';
		fb_edit_mfps_bestuecken_z.st_config.b_config_fertig := TRUE;
		
		fb_edit_mfps_bestuecken_y.st_config.b_config_fertig := FALSE;
		fb_edit_mfps_bestuecken_y.st_config.b_station_aktiv := TRUE;
		fb_edit_mfps_bestuecken_y.st_config.i16_meld_startindex := 660;
		fb_edit_mfps_bestuecken_y.st_config.str_beschreibung := ' ';
		fb_edit_mfps_bestuecken_y.st_config.str_instanz_name := 'Kurvenscheibeneditor Bestücken Y-Achse';
		fb_edit_mfps_bestuecken_y.st_config.b_config_fertig := TRUE;
		
		fb_edit_mfps_yz_tisch.st_config.b_config_fertig := FALSE;
		fb_edit_mfps_yz_tisch.st_config.b_station_aktiv := TRUE;
		fb_edit_mfps_yz_tisch.st_config.i16_meld_startindex := 680;
		fb_edit_mfps_yz_tisch.st_config.str_beschreibung := ' ';
		fb_edit_mfps_yz_tisch.st_config.str_instanz_name := 'Kurvenscheibeneditor YZ-Tisch';
		fb_edit_mfps_yz_tisch.st_config.b_config_fertig := TRUE;

